(* CODESYS project CtaDevClimaVeneta_1.0.0.0.library
   Description: CtaDevClimaVeneta Library für ClimaVeneta Modbus auslesung
   Version: 1.0.0.0
   Title: CtaDevClimaVeneta
   Author: SIS
   Company: CTA
   DocFormat: reStructuredText
   Placeholder: CtaDevClimaVeneta
   CompiledLibraryCompatibilityVersion: CODESYS V3.5 SP16 Patch 3
   LanguageModelAttribute: qualified-access-only
   DefaultNamespace: CtaDevClimaVeneta

Project tree, tasks and I/O mapping:
  libraries: CtaAppBmk, 2.0.0.1 (CTA); CtaAppReport, 2.0.0.2 (CTA); CtaAppInfluxLog, 1.0.0.1 (CTA); Standard, 3.5.18.0 (System); CtaAppRefrigants, 1.0.0.0 (CTA); CtaAppModbus, 2.0.0.3 (CTA)
  40 Visualizations/
  30 Program Organization Units/
    MODBUS_FB_CLIMAVENETA/
      function block MODBUS_CLIMAVENETA [ST]: COM_DATA
      text list txtAlamsW3000
      text list txtWpReport
  00000000-0000-0000-0000-000000000000|D:\CoDeSys\LibrariesV3\trunk\Intern\CAA\CAA Template\3.4.0.0 draft\Placeholder.xml
  00000000-0000-0000-0000-000000000000|D:\CoDeSys\LibrariesV3\trunk\Intern\CAA\CAA Template\3.2.0.3 draft\Prefix.pdf
  00000000-0000-0000-0000-000000000000|D:\CoDeSys\LibrariesV3\trunk\Intern\CAA\CAA Template\3.5.2.0 draft\Placeholder.xml
  20 Structs/
  50 Images/
  10 Documenation/
    global variables VersionHistory
    global variables readMe
  21 Interface/
  11 Library Parameter/
  12 Konstanten/
  60 Textlisten/
  13 Globale Variablen/
*)

// 10 Documenation/VersionHistory
(* 

.. image:: ../../Images/CTA_Logo.jpg
   :align: right
   :width: 15% 

**Vorlage**   


============ =========== =========== ============================================
**Date**     **Version** **Author**  **Change**
------------ ----------- ----------- --------------------------------------------
22.07.2026   1.0.0.0     SIS         Bibliothek erstellt

============ =========== =========== ============================================


*)
VAR_GLOBAL
    stInfo : STRING:= '0.0.0.0, CtaDevClimaVeneta, CTA';
END_VAR

// 10 Documenation/readMe
(*
**ReadMe**

 
 |  Diese Bibliothek dient der standartisierten auslesung von Climaveneta Maschinen
 |     
*)

VAR_GLOBAL
    xReadMeDone              :   BOOL;
END_VAR

// 30 Program Organization Units/MODBUS_FB_CLIMAVENETA/MODBUS_CLIMAVENETA
FUNCTION_BLOCK MODBUS_CLIMAVENETA
VAR CONSTANT
	stTxtReportError		:	STRING											:= 'CtaDevClimaVeneta.txtWpReport';
END_VAR
VAR_INPUT
	ITF_BMK					:	CtaAppBmk.ITF_BMK;
	ITF_REPORTMANAGER		:	CtaAppReport.ITF_REPORTMANAGER;
	set_point				:	REAL;											// Sollwert
	_rBeschränkung			:	REAL;											// Demand Limit
	_xBeschränkungEN		:	BOOL;											// Demand Limit enable
END_VAR
VAR_OUTPUT
	_xModBusError			:	BOOL;
	_v1k1_on				:	BOOL;
	_v1k2_on				:	BOOL;	
	_v2k1_on				:	BOOL;
	_v2k2_on				:	BOOL;	
	_xAlarm1V1				:	BOOL;
	_xAlarm1V2				:	BOOL;
	_xAlarm1V3				:	BOOL;
	_xAlarm1V4				:	BOOL;
	
	_rHochdruckV1			:	REAL;
	_rHochdruckTempV1		:	REAL;
	_rHochdruckV2			:	REAL;
	_rHochdruckTempV2		:	REAL;
	
	_rNiederdruckV1			:	REAL;
	_rNiederdruckTempV1		:	REAL;
	_rNiederdruckV2			:	REAL;
	_rNiederdruckTempV2		:	REAL;

	_rFehlerCode			:	REAL;
	
END_VAR
VAR
	_ayMbData				:	ARRAY[0..16] OF WORD;
	_ayTrendLogBool			:	ARRAY[1..15] OF CtaAppInfluxLog.FB_LOG_NODE_BOOL;
	_ayTrendLogReal			:	ARRAY[1..15] OF CtaAppInfluxLog.FB_LOG_NODE_REAL;
	_ayReports				:	ARRAY[0..00] OF CtaAppReport.fbReporter;
	_ayMbDataBOOL			:	ARRAY[0..16] OF BOOL;
END_VAR

IF __QUERYINTERFACE(ITF_BMK,ITF_BMK) THEN

	_ayTrendLogReal[01].ENABLE 		:= TRUE;
	_ayTrendLogReal[01].KEY	 		:= CONCAT(ITF_BMK.proGetBMK,'_rHochdruckV1');
	_ayTrendLogReal[01].SET_VALUE	:= _rHochdruckV1;
	
	_ayTrendLogReal[02].ENABLE 		:= TRUE;
	_ayTrendLogReal[02].KEY	 		:= CONCAT(ITF_BMK.proGetBMK,'_rHochdruckV2');
	_ayTrendLogReal[02].SET_VALUE	:= _rHochdruckV2;

	_ayTrendLogReal[03].ENABLE 		:= TRUE;
	_ayTrendLogReal[03].KEY	 		:= CONCAT(ITF_BMK.proGetBMK,'_rNiederdruckV1');
	_ayTrendLogReal[03].SET_VALUE	:= _rNiederdruckV1;
	
	_ayTrendLogReal[04].ENABLE 		:= TRUE;
	_ayTrendLogReal[04].KEY	 		:= CONCAT(ITF_BMK.proGetBMK,'_rNiederdruckV2');
	_ayTrendLogReal[04].SET_VALUE	:= _rNiederdruckV2;
	
	_ayTrendLogReal[05].ENABLE 		:= TRUE;
	_ayTrendLogReal[05].KEY	 		:= CONCAT(ITF_BMK.proGetBMK,'_rFehlerCode');
	_ayTrendLogReal[05].SET_VALUE	:= _rFehlerCode;
	
	_ayTrendLogReal[06].ENABLE 		:= TRUE;
	_ayTrendLogReal[06].KEY	 		:= CONCAT(ITF_BMK.proGetBMK,'_rHochdruckTempV1');
	_ayTrendLogReal[06].SET_VALUE	:= _rHochdruckTempV1;
	
	_ayTrendLogReal[07].ENABLE 		:= TRUE;
	_ayTrendLogReal[07].KEY	 		:= CONCAT(ITF_BMK.proGetBMK,'_rHochdruckTempV2');
	_ayTrendLogReal[07].SET_VALUE	:= _rHochdruckTempV2;
	
	_ayTrendLogReal[08].ENABLE 		:= TRUE;
	_ayTrendLogReal[08].KEY	 		:= CONCAT(ITF_BMK.proGetBMK,'_rNiederdruckTempV1');
	_ayTrendLogReal[08].SET_VALUE	:= _rNiederdruckTempV1;
	
	_ayTrendLogReal[09].ENABLE 		:= TRUE;
	_ayTrendLogReal[09].KEY	 		:= CONCAT(ITF_BMK.proGetBMK,'_rNiederdruckTempV2');
	_ayTrendLogReal[09].SET_VALUE	:= _rNiederdruckTempV2;

	_ayTrendLogBool[05].ENABLE 		:= TRUE;
	_ayTrendLogBool[05].KEY	 		:= CONCAT(ITF_BMK.proGetBMK,'_xAlarm1V1');
	_ayTrendLogBool[05].SET_VALUE	:= _xAlarm1V1;

	_ayTrendLogBool[06].ENABLE 		:= TRUE;
	_ayTrendLogBool[06].KEY	 		:= CONCAT(ITF_BMK.proGetBMK,'_xAlarm1V2');
	_ayTrendLogBool[06].SET_VALUE	:= _xAlarm1V2;

	_ayTrendLogBool[07].ENABLE 		:= TRUE;
	_ayTrendLogBool[07].KEY	 		:= CONCAT(ITF_BMK.proGetBMK,'_xAlarm1V3');
	_ayTrendLogBool[07].SET_VALUE	:= _xAlarm1V3;

	_ayTrendLogBool[08].ENABLE 		:= TRUE;
	_ayTrendLogBool[08].KEY	 		:= CONCAT(ITF_BMK.proGetBMK,'_xAlarm1V4');
	_ayTrendLogBool[08].SET_VALUE	:= _xAlarm1V4;	
	
	(* Rechnung Bar zu Temp *)
	_rHochdruckTempV1 	:= CtaAppRefrigants.fcPressToTemp_UserDefined(_rHochdruckV1,CtaAppRefrigants.GVL_REFRIGANTS.FB_COURRENT_REFRIGANT.enGasType,FALSE);
	_rNiederdruckTempV1 := CtaAppRefrigants.fcPressToTemp_UserDefined(_rNiederdruckV1,CtaAppRefrigants.GVL_REFRIGANTS.FB_COURRENT_REFRIGANT.enGasType,FALSE);
	
	_rHochdruckTempV2	:= CtaAppRefrigants.fcPressToTemp_UserDefined(_rHochdruckV2,CtaAppRefrigants.GVL_REFRIGANTS.FB_COURRENT_REFRIGANT.enGasType,FALSE);
	_rNiederdruckTempV2 := CtaAppRefrigants.fcPressToTemp_UserDefined(_rNiederdruckV2,CtaAppRefrigants.GVL_REFRIGANTS.FB_COURRENT_REFRIGANT.enGasType,FALSE);

	IF __QUERYINTERFACE(ITF_REPORTMANAGER,ITF_REPORTMANAGER) THEN
		_ayReports[0].metReport(	xSetReportIn				:=	_xModBusError,
									iReportID					:=  60,
									enReportTypeIn				:=  CtaAppReport.enReportType.Error,
									enReportAcknowledgeTypeIn	:=	CtaAppReport.enReportacknowledgeType.Auto,
									tDelay						:=	T#1M,
									ITF_BMK_IN					:=  ITF_BMK,
									pstReportTextListIn			:=  ADR(stTxtReportError),
									stOptionalReportText		:=  '',
									iRetryTilReportLock			:=  3,
									xResetCount					:=  FALSE,
									tReset						:=  T#24H);
		ITF_REPORTMANAGER.metSyncReporter(_ayReports[0]);
	END_IF;
END_IF;

METHOD COM_DATA
VAR_INPUT
	ITF_MB_CLIENT		:	CtaAppModbus.ITF_CLIENT;
END_VAR
VAR 
	ITF_MB_CLIENT_TCP	:	CtaAppModbus.ITF_MB_CLIENT_TCP;
	ITF_MB_CLIENT_RTU	:	CtaAppModbus.ITF_MB_CLIENT_RTU;
	offset				: 	INT;
END_VAR
// Modbus TCP
IF __QUERYINTERFACE(ITF_MB_CLIENT, ITF_MB_CLIENT_TCP ) THEN	
	// Delet rtu
	IF __QUERYINTERFACE(ITF_MB_CLIENT_RTU, ITF_MB_CLIENT_RTU ) THEN
		ITF_MB_CLIENT_RTU.DESTROY_ALL_JOBS_REQUEST();
		ITF_MB_CLIENT_RTU := 0;
	END_IF;
	
	_xModBusError := ITF_MB_CLIENT_TCP.ERROR;
	offset		  := -1;	
	
	// High pressure transducer
	ITF_MB_CLIENT_TCP.CREATE_JOB( _byMbFunction := 04 ,	_wMbAdress := TO_WORD(  13 + offset ), _pData := ADR(_ayMbData[00]), _wQuantity := 1); _rHochdruckV1				:= TO_REAL(TO_INT(_ayMbData[00])) / 10 ;
	ITF_MB_CLIENT_TCP.CREATE_JOB( _byMbFunction := 04 ,	_wMbAdress := TO_WORD(  14 + offset ), _pData := ADR(_ayMbData[01]), _wQuantity := 1); _rHochdruckV2				:= TO_REAL(TO_INT(_ayMbData[01])) / 10 ;
     
	// Low pressure transducer                                                                
	ITF_MB_CLIENT_TCP.CREATE_JOB( _byMbFunction := 04 ,	_wMbAdress := TO_WORD(  17 + offset ), _pData := ADR(_ayMbData[02]), _wQuantity := 1); _rNiederdruckV1			:= TO_REAL(TO_INT(_ayMbData[02])) / 10 ;
	ITF_MB_CLIENT_TCP.CREATE_JOB( _byMbFunction := 04 ,	_wMbAdress := TO_WORD(  18 + offset ), _pData := ADR(_ayMbData[03]), _wQuantity := 1); _rNiederdruckV2			:= TO_REAL(TO_INT(_ayMbData[03])) / 10 ;
        
	// Compressor status                                                            
	ITF_MB_CLIENT_TCP.CREATE_JOB( _byMbFunction := 04 ,	_wMbAdress := TO_WORD(5017 + offset ), _pData := ADR(_ayMbData[04]), _wQuantity := 1); _xAlarm1V1	 		:= _ayMbData[04].04;	_v1k1_on		:= _ayMbData[04].2;	
	ITF_MB_CLIENT_TCP.CREATE_JOB( _byMbFunction := 04 ,	_wMbAdress := TO_WORD(5018 + offset ), _pData := ADR(_ayMbData[05]), _wQuantity := 1); _xAlarm1V2	 		:= _ayMbData[05].04;	_v1k2_on		:= _ayMbData[05].2;	
	ITF_MB_CLIENT_TCP.CREATE_JOB( _byMbFunction := 04 ,	_wMbAdress := TO_WORD(5019 + offset ), _pData := ADR(_ayMbData[06]), _wQuantity := 1); _xAlarm1V3	 		:= _ayMbData[06].04;	_v2k1_on		:= _ayMbData[06].2;	 
	ITF_MB_CLIENT_TCP.CREATE_JOB( _byMbFunction := 04 ,	_wMbAdress := TO_WORD(5020 + offset ), _pData := ADR(_ayMbData[07]), _wQuantity := 1); _xAlarm1V4	 		:= _ayMbData[07].04;	_v2k2_on		:= _ayMbData[07].2;
	
	// Active alarm code (with greater priority)                                                                     
	ITF_MB_CLIENT_TCP.CREATE_JOB( _byMbFunction := 04 ,	_wMbAdress := TO_WORD(5034 + offset ), _pData := ADR(_ayMbData[09]), _wQuantity := 1); _rFehlerCode		:= TO_REAL(TO_INT(_ayMbData[09]))  ;

	// Temperature controller limitation in heat pump
	_ayMbData[12] := TO_WORD(TO_INT(_rBeschränkung * 10));
	ITF_MB_CLIENT_TCP.CREATE_JOB( _byMbFunction := 06, 	_wMbAdress := TO_WORD(5046 + offset ), _pData := ADR(_ayMbData[12]), _wQuantity := 1)  ; 
	
	
	_ayMbDataBOOL[00] := _xBeschränkungEN;
	ITF_MB_CLIENT_TCP.CREATE_JOB( _byMbFunction := 05 ,	_wMbAdress := TO_WORD( 284 + offset ), _pData := ADR(_ayMbDataBOOL[00]), _wQuantity := 1);
	
	// Chiller temperature setpoint 
	_ayMbData[13] := TO_WORD(TO_INT(set_point * 10));
	ITF_MB_CLIENT_TCP.CREATE_JOB( _byMbFunction := 06 , _wMbAdress := TO_WORD( 	 2 + offset ), _pData := ADR(_ayMbData[13]), _wQuantity := 1)  ; 
	
// Modbus RTU
ELSIF __QUERYINTERFACE(ITF_MB_CLIENT, ITF_MB_CLIENT_RTU ) THEN	
	// Delet tcp
	IF __QUERYINTERFACE(ITF_MB_CLIENT_TCP, ITF_MB_CLIENT_TCP ) THEN
		ITF_MB_CLIENT_TCP.DESTROY_ALL_JOBS_REQUEST();
		ITF_MB_CLIENT_TCP := 0;
	END_IF;
	
	_xModBusError := ITF_MB_CLIENT_RTU.ERROR;
	offset		  := 0;		
	
	// High pressure transducer
	ITF_MB_CLIENT_RTU.CREATE_JOB( _byMbFunction := 04 ,	_wMbAdress :=   12 , _pData := ADR(_ayMbData[00]), _wQuantity := 1); _rHochdruckV1				:= TO_REAL(TO_INT(_ayMbData[00])) / 10 ;
	ITF_MB_CLIENT_RTU.CREATE_JOB( _byMbFunction := 04 ,	_wMbAdress :=   13 , _pData := ADR(_ayMbData[01]), _wQuantity := 1); _rHochdruckV2				:= TO_REAL(TO_INT(_ayMbData[01])) / 10 ;
	
	// Low pressure transducer
	ITF_MB_CLIENT_RTU.CREATE_JOB( _byMbFunction := 04 ,	_wMbAdress :=   16 , _pData := ADR(_ayMbData[02]), _wQuantity := 1); _rNiederdruckV1			:= TO_REAL(TO_INT(_ayMbData[02])) / 10 ;
	ITF_MB_CLIENT_RTU.CREATE_JOB( _byMbFunction := 04 ,	_wMbAdress :=   17 , _pData := ADR(_ayMbData[03]), _wQuantity := 1); _rNiederdruckV2			:= TO_REAL(TO_INT(_ayMbData[03])) / 10 ;

	// Compressor status
	ITF_MB_CLIENT_RTU.CREATE_JOB( _byMbFunction := 04 ,	_wMbAdress :=  143 , _pData := ADR(_ayMbData[04]), _wQuantity := 1); _xAlarm1V1	 		:= _ayMbData[04].04;	_v1k1_on		:= _ayMbData[04].2;	
	ITF_MB_CLIENT_RTU.CREATE_JOB( _byMbFunction := 04 ,	_wMbAdress :=  144 , _pData := ADR(_ayMbData[05]), _wQuantity := 1); _xAlarm1V2	 		:= _ayMbData[05].04;	_v1k2_on		:= _ayMbData[05].2;	
	ITF_MB_CLIENT_RTU.CREATE_JOB( _byMbFunction := 04 ,	_wMbAdress :=  145 , _pData := ADR(_ayMbData[06]), _wQuantity := 1); _xAlarm1V3	 		:= _ayMbData[06].04;	_v2k1_on		:= _ayMbData[06].2;	 
	ITF_MB_CLIENT_RTU.CREATE_JOB( _byMbFunction := 04 ,	_wMbAdress :=  146 , _pData := ADR(_ayMbData[07]), _wQuantity := 1); _xAlarm1V4	 		:= _ayMbData[07].04;	_v2k2_on		:= _ayMbData[07].2;
	
	// Active alarm code (with greater priority) 
	ITF_MB_CLIENT_RTU.CREATE_JOB( _byMbFunction := 04 ,	_wMbAdress :=  160 , _pData := ADR(_ayMbData[09]), _wQuantity := 1); _rFehlerCode		:= TO_REAL(TO_INT(_ayMbData[09]))  ;

	// Temperature controller limitation in heat pump
	_ayMbData[12] := TO_WORD(TO_INT(_rBeschränkung * 10));
	ITF_MB_CLIENT_RTU.CREATE_JOB( _byMbFunction := 06, 	_wMbAdress :=  172, _pData := ADR(_ayMbData[12]), _wQuantity := 1)  ; 
	
	_ayMbDataBOOL[00] := _xBeschränkungEN;
	ITF_MB_CLIENT_RTU.CREATE_JOB( _byMbFunction := 05 ,	_wMbAdress :=   33 , _pData := ADR(_ayMbDataBOOL[00]), _wQuantity := 1);
	
	// Chiller temperature setpoint 
	_ayMbData[13] := TO_WORD(TO_INT(set_point * 10));
	ITF_MB_CLIENT_RTU.CREATE_JOB( _byMbFunction := 06 , _wMbAdress :=  	 1, _pData := ADR(_ayMbData[13]), _wQuantity := 1)  ; 
	

ELSE
	_xModBusError := TRUE;
END_IF;
END_METHOD

END_FUNCTION_BLOCK

(* text list txtAlamsW3000 (id | default | de | en | fr | it)
  2 | Phasensequenz / Spannung außer Bereich | Phasensequenz / Spannung außer Bereich | Phase sequence / voltage out of range | Séquence de phases / tension hors plage | Sequenza di fase / tensione fuori intervallo
  3 | Kein Wasserfluss am Verdampfer | Kein Wasserfluss am Verdampfer | No water flow at evaporator | No water flow at évaporateur | No water flow at evaporatore
  5 | Niedrige Temperatur am Eingang | Niedrige Temperatur am Eingang | Low temperature am inlet | Low temperature am entrée | Low temperature am ingresso
  6 | Hohe Temperatur am Eingang | Hohe Temperatur am Eingang | High temperature am inlet | High temperature am entrée | High temperature am ingresso
  7 | Blockierung alternative Quelle der Anlage | Blockierung alternative Quelle der Anlage | Lockout: plant alternative source | Blocage : source alternative de l’installation | Blocco: fonte alternativa dell’impianto
  8 | Blockierung alternative DHW -quelle | Blockierung alternative DHW -quelle | Lockout: alternative DHW source | Blocage : source ECS (DHW) alternative | Blocco: sorgente ACS alternativa
  10 | Frostschutz Verdampfer Niedrige Wassertemperatur am Verdampferausgang. Es wird außerdem angezeigt, für welchen Verdampfer der Alarm gilt (bei mehr als einem Verdampfer). Der Alarm tritt auch dann auf, wenn die Frostschutz - Begrenzung in einem Zeitraum von 8 Betriebsstunden öfter als 5 -mal ausgelöst wird. M CI STG0073 | Frostschutz Verdampfer Niedrige Wassertemperatur am Verdampferausgang. Es wird außerdem angezeigt, für welchen Verdampfer der Alarm gilt (bei mehr als einem Verdampfer). Der Alarm tritt auch dann auf, wenn die Frostschutz - Begrenzung in einem Zeitraum von 8 Betriebsstunden öfter als 5 -mal ausgelöst wird. M CI STG0073 | Frost protection evaporator Niedrige Wassertemperatur am evaporatoroutlet. Es wird außerdem angezeigt, für welchen evaporator Alarm gilt (bei mehr als einem evaporator). Alarm tritt auch dann auf, wenn Frostschutz - Begrenzung in einem Zeitraum von 8 Betriebsstunden öfter als 5 -mal ausgelöst wird. M CI STG0073 | Frost protection évaporateur Niedrige Wassertemperatur am évaporateursortie. Es wird außerdem angezeigt, für welchen évaporateur Alarm gilt (bei mehr als einem évaporateur). Alarm tritt auch dann auf, wenn Frostschutz - Begrenzung in einem Zeitraum von 8 Betriebsstunden öfter als 5 -mal ausgelöst wird. M CI STG0073 | Frost protection evaporatore Niedrige Wassertemperatur am evaporatoreuscita. Es wird außerdem angezeigt, für welchen evaporatore Alarm gilt (bei mehr als einem evaporatore). Alarm tritt auch dann auf, wenn Frostschutz - Begrenzung in einem Zeitraum von 8 Betriebsstunden öfter als 5 -mal ausgelöst wird. M CI STG0073
  14 | Unzureichender Anlagendruck | Unzureichender Anlagendruck | Insufficient system pressure | Pression système insuffisante | Pressione impianto insufficiente
  17 | Niedrige Außenlufttemperatur | Niedrige Außenlufttemperatur | Low outdoor air temperature | Température extérieure basse | Temperatura aria esterna bassa
  21 | Geringe Wassermenge in der Anlage | Geringe Wassermenge in der Anlage | Low water content in system | Faible volume d’eau dans l’installation | Basso contenuto d’acqua nel sistema
  22 | Niedriger Wasserdurchfluss in der Anlage | Niedriger Wasserdurchfluss in der Anlage | Low water flow in system | Low water flow in installation | Low water flow in impianto
  23 | Hoher Wasserdurchfluss | Hoher Wasserdurchfluss | High water flow | Débit d’eau élevé | Portata d’acqua elevata
  41 | Niedrige Temperatur am Verflüssigereingang | Niedrige Temperatur am Verflüssigereingang | Low temperature at condenser inlet | Low temperature at condenser inlet | Low temperature at condenser inlet
  42 | Hohe Temperatur am Verflüssigerausgang | Hohe Temperatur am Verflüssigerausgang | High temperature at condenser outlet | High temperature at condenser outlet | High temperature at condenser outlet
  43 | Niedriger Wasserdurchfluss im Verflüssiger | Niedriger Wasserdurchfluss im Verflüssiger | Low water flow im condenser | Low water flow im condenseur | Low water flow im condensatore
  44 | Hoher Wasserdurchfluss im Verflüssiger | Hoher Wasserdurchfluss im Verflüssiger | High water flow | Débit d’eau élevé | Portata d’acqua elevata
  45 | Kein Wasserfluss am Verflüssiger „Kein Wasserfluss am Verdampfer” (nur bei Wasser/Wasser -Einheiten mit Freon -Umkehr). A/M U | Kein Wasserfluss am Verflüssiger „Kein Wasserfluss am Verdampfer” (nur bei Wasser/Wasser -Einheiten mit Freon -Umkehr). A/M U | No water flow at condenser „No water flow at evaporator” (nur bei Wasser/Wasser -uniten mit Freon -Umkehr). A/M U | No water flow at condenseur „No water flow at évaporateur” (nur bei Wasser/Wasser -unitéen mit Freon -Umkehr). A/M U | No water flow at condensatore „No water flow at evaporatore” (nur bei Wasser/Wasser -unitàen mit Freon -Umkehr). A/M U
  46 | Kein Wasserfluss am WRG | Kein Wasserfluss am WRG | No water flow at heat recovery | No water flow at récupération de chaleur | No water flow at recupero di calore
  50 | Totalausfall Kältemaschine  | Totalausfall Kältemaschine  | Complete failure of the cooling system | Panne complète du système de refroidissement | Guasto completo della macchina frigorifera
  51 | Wartung Pumpe 1 | Wartung Pumpe 1 | Maintenance pump 1 | Maintenance pompe 1 | Maintenance pompa 1
  57 | Wartung WRG/DHW -Pumpe (Bei Einheiten mit WRG -Pumpe) Die Grenze der zulässigen Stunden der WRG -Pumpe wurde überschritten. S - STG0007 | Wartung WRG/DHW -Pumpe (Bei Einheiten mit WRG -Pumpe) Die Grenze der zulässigen Stunden der WRG -Pumpe wurde überschritten. S - STG0007 | Maintenance heat recovery/DHW -pump (Bei uniten mit heat recovery -pump) Grenze zulässigen Stunden heat recovery -pump wurde überschritten. S - STG0007 | Maintenance récupération de chaleur/DHW -pompe (Bei unitéen mit récupération de chaleur -pompe) Grenze zulässigen Stunden récupération de chaleur -pompe wurde überschritten. S - STG0007 | Maintenance recupero di calore/DHW -pompa (Bei unitàen mit recupero di calore -pompa) Grenze zulässigen Stunden recupero di calore -pompa wurde überschritten. S - STG0007
  58 | Wartung Verflüssigerpumpe (Bei Einheiten mit Verflüssigerpumpe) Die Grenze der zulässigen Stunden der Verflüssigerpumpe wurde überschritten. S - STG0010 | Wartung Verflüssigerpumpe (Bei Einheiten mit Verflüssigerpumpe) Die Grenze der zulässigen Stunden der Verflüssigerpumpe wurde überschritten. S - STG0010 | Maintenance condenserpump (Bei uniten mit condenserpump) Grenze zulässigen Stunden condenserpump wurde überschritten. S - STG0010 | Maintenance condenseurpompe (Bei unitéen mit condenseurpompe) Grenze zulässigen Stunden condenseurpompe wurde überschritten. S - STG0010 | Maintenance condensatorepompa (Bei unitàen mit condensatorepompa) Grenze zulässigen Stunden condensatorepompa wurde überschritten. S - STG0010
  61 | Offline Driver Unterkühlung / erste Stufe Nr.1 | Offline Driver Unterkühlung / erste Stufe Nr.1 | Offline Driver Unterkühlung / erste Stufe Nr.1 | Offline Driver Unterkühlung / erste Stufe Nr.1 | Offline Driver Unterkühlung / erste Stufe Nr.1
  62 | Offline Driver Unterkühlung / erste Stufe Nr.2 „Wie oben, für den Kreislauf Nr.2“ / Ventil erste Stufe des Verdichters 2. A CI | Offline Driver Unterkühlung / erste Stufe Nr.2 „Wie oben, für den Kreislauf Nr.2“ / Ventil erste Stufe des Verdichters 2. A CI | Offline Driver Unterkühlung / erste Stufe Nr.2 „Wie oben, für circuit Nr.2“ / Ventil erste Stufe compressors 2. A CI | Offline Driver Unterkühlung / erste Stufe Nr.2 „Wie oben, für circuit Nr.2“ / Ventil erste Stufe compresseurs 2. A CI | Offline Driver Unterkühlung / erste Stufe Nr.2 „Wie oben, für circuito Nr.2“ / Ventil erste Stufe compressores 2. A CI
  63 | Offline Driver Unterkühlung / erste Stufe Nr.3 „Wie oben, für den Kreislauf Nr.1“ / Ventil erste Stufe des Verdichters 3. A CI | Offline Driver Unterkühlung / erste Stufe Nr.3 „Wie oben, für den Kreislauf Nr.1“ / Ventil erste Stufe des Verdichters 3. A CI | Offline Driver Unterkühlung / erste Stufe Nr.3 „Wie oben, für circuit Nr.1“ / Ventil erste Stufe compressors 3. A CI | Offline Driver Unterkühlung / erste Stufe Nr.3 „Wie oben, für circuit Nr.1“ / Ventil erste Stufe compresseurs 3. A CI | Offline Driver Unterkühlung / erste Stufe Nr.3 „Wie oben, für circuito Nr.1“ / Ventil erste Stufe compressores 3. A CI
  64 | Offline Driver Unterkühlung / erste Stufe Nr.4 „Wie oben, für den Kreislauf Nr.2“ / Ventil erste Stufe des Verdichters 4. A CI | Offline Driver Unterkühlung / erste Stufe Nr.4 „Wie oben, für den Kreislauf Nr.2“ / Ventil erste Stufe des Verdichters 4. A CI | Offline Driver Unterkühlung / erste Stufe Nr.4 „Wie oben, für circuit Nr.2“ / Ventil erste Stufe compressors 4. A CI | Offline Driver Unterkühlung / erste Stufe Nr.4 „Wie oben, für circuit Nr.2“ / Ventil erste Stufe compresseurs 4. A CI | Offline Driver Unterkühlung / erste Stufe Nr.4 „Wie oben, für circuito Nr.2“ / Ventil erste Stufe compressores 4. A CI
  65 | Niedrige Wassermenge im Wärmerückgewinnungskreislauf | Niedrige Wassermenge im Wärmerückgewinnungskreislauf | Niedrige Wassermenge im heat recovery circuit | Niedrige Wassermenge im circuit de récupération de chaleur | Niedrige Wassermenge im circuit di recupero di calore
  66 | Niedriger Wasserdurchfluss im Wärmerückgewinnungskreislauf | Niedriger Wasserdurchfluss im Wärmerückgewinnungskreislauf | Low water flow im heat recovery circuit | Low water flow im circuit de récupération de chaleur | Low water flow im circuit di recupero di calore
  67 | Alarm Antilegionellenfunktion | Alarm Antilegionellenfunktion | Alarm Antilegionellenfunktion | Alarm Antilegionellenfunktion | Alarm Antilegionellenfunktion
  68 | Störung von Steuerung Kühlteil Meldet einen von der Hauptreglereinheit kommenden Alarm in den Einheiten mit +2P -Modul. Um den Alarm im Detail anzuzeigen und rückzustellen, muss mit der Tastenkombination [ESC+UP] zur Schnittstelle der Hauptreglereinheit übergegangen werden. S - | Störung von Steuerung Kühlteil Meldet einen von der Hauptreglereinheit kommenden Alarm in den Einheiten mit +2P -Modul. Um den Alarm im Detail anzuzeigen und rückzustellen, muss mit der Tastenkombination [ESC+UP] zur Schnittstelle der Hauptreglereinheit übergegangen werden. S - | Fault von Steuerung Kühlteil Meldet einen von Hauptreglerunit kommenden Alarm in uniten mit +2P -Modul. Um Alarm im Detail anzuzeigen und rückzustellen, muss mit Tastenkombination [ESC+UP] zur Schnittstelle Hauptreglerunit übergegangen werden. S - | Fault von Steuerung Kühlteil Meldet einen von Hauptreglerunité kommenden Alarm in unitéen mit +2P -Modul. Um Alarm im Detail anzuzeigen und rückzustellen, muss mit Tastenkombination [ESC+UP] zur Schnittstelle Hauptreglerunité übergegangen werden. S - | Fault von Steuerung Kühlteil Meldet einen von Hauptreglerunità kommenden Alarm in unitàen mit +2P -Modul. Um Alarm im Detail anzuzeigen und rückzustellen, muss mit Tastenkombination [ESC+UP] zur Schnittstelle Hauptreglerunità übergegangen werden. S -
  69 | Störung von Steuerung Luftteil Meldet einen von der Steuerung des Luftteils kommenden Alarm in den Rooftop -Einheiten. Um den Alarm im Detail anzuzeigen und rückzustellen, muss mit der Tastenkombination [ESC+UP] zur Schnittstelle der Hauptreglereinheit übergegangen werden. S - | Störung von Steuerung Luftteil Meldet einen von der Steuerung des Luftteils kommenden Alarm in den Rooftop -Einheiten. Um den Alarm im Detail anzuzeigen und rückzustellen, muss mit der Tastenkombination [ESC+UP] zur Schnittstelle der Hauptreglereinheit übergegangen werden. S - | Fault von Steuerung Luftteil Meldet einen von Steuerung Luftteils kommenden Alarm in Rooftop -uniten. Um Alarm im Detail anzuzeigen und rückzustellen, muss mit Tastenkombination [ESC+UP] zur Schnittstelle Hauptreglerunit übergegangen werden. S - | Fault von Steuerung Luftteil Meldet einen von Steuerung Luftteils kommenden Alarm in Rooftop -unitéen. Um Alarm im Detail anzuzeigen und rückzustellen, muss mit Tastenkombination [ESC+UP] zur Schnittstelle Hauptreglerunité übergegangen werden. S - | Fault von Steuerung Luftteil Meldet einen von Steuerung Luftteils kommenden Alarm in Rooftop -unitàen. Um Alarm im Detail anzuzeigen und rückzustellen, muss mit Tastenkombination [ESC+UP] zur Schnittstelle Hauptreglerunità übergegangen werden. S -
  70 | Störung von Steuerung +2P -Modul Meldet einen von der Reglereinheit kommenden Alarm des Moduls +2P. Um den Alarm im Detail anzuzeigen und rückzustellen, muss mit der Tastenkombination [ESC+UP] zur Schnittstelle der Reglereinheit +2P übergegangen werden. S - | Störung von Steuerung +2P -Modul Meldet einen von der Reglereinheit kommenden Alarm des Moduls +2P. Um den Alarm im Detail anzuzeigen und rückzustellen, muss mit der Tastenkombination [ESC+UP] zur Schnittstelle der Reglereinheit +2P übergegangen werden. S - | Fault von Steuerung +2P -Modul Meldet einen von Reglerunit kommenden Alarm Moduls +2P. Um Alarm im Detail anzuzeigen und rückzustellen, muss mit Tastenkombination [ESC+UP] zur Schnittstelle Reglerunit +2P übergegangen werden. S - | Fault von Steuerung +2P -Modul Meldet einen von Reglerunité kommenden Alarm Moduls +2P. Um Alarm im Detail anzuzeigen und rückzustellen, muss mit Tastenkombination [ESC+UP] zur Schnittstelle Reglerunité +2P übergegangen werden. S - | Fault von Steuerung +2P -Modul Meldet einen von Reglerunità kommenden Alarm Moduls +2P. Um Alarm im Detail anzuzeigen und rückzustellen, muss mit Tastenkombination [ESC+UP] zur Schnittstelle Reglerunità +2P übergegangen werden. S -
  72 | Hoher Wasserdurchfluss im Wärmerückgewinnungskreislauf | Hoher Wasserdurchfluss im Wärmerückgewinnungskreislauf | High water flow | Débit d’eau élevé | Portata d’acqua elevata
  75 | Frostschutz Verflüssiger Niedrige Wassertemperatur am Ausgang des Verflüssigers. Mit Ausnahme von W3000+ Basis wird außerdem angegeben, welcher Verflüssiger (bei mehr als einem) von dem Alarm betroffen ist. Der Alarm tritt auch dann auf, wenn die Frostschutzfunktion mehr als 5 -mal innerhalb von 8 Betriebsstunden ausgelöst wird (nur bei Wasser/Wasser -Einheiten mit Freon -Umkehr). M U* STG0077 | Frostschutz Verflüssiger Niedrige Wassertemperatur am Ausgang des Verflüssigers. Mit Ausnahme von W3000+ Basis wird außerdem angegeben, welcher Verflüssiger (bei mehr als einem) von dem Alarm betroffen ist. Der Alarm tritt auch dann auf, wenn die Frostschutzfunktion mehr als 5 -mal innerhalb von 8 Betriebsstunden ausgelöst wird (nur bei Wasser/Wasser -Einheiten mit Freon -Umkehr). M U* STG0077 | Frost protection condenser Niedrige Wassertemperatur am outlet condensers. Mit Ausnahme von W3000+ Basis wird außerdem angegeben, welcher condenser (bei mehr als einem) von Alarm betroffen ist. Alarm tritt auch dann auf, wenn Frostschutzfunktion mehr als 5 -mal innerhalb von 8 Betriebsstunden ausgelöst wird (nur bei Wasser/Wasser -uniten mit Freon -Umkehr). M U* STG0077 | Frost protection condenseur Niedrige Wassertemperatur am sortie condenseurs. Mit Ausnahme von W3000+ Basis wird außerdem angegeben, welcher condenseur (bei mehr als einem) von Alarm betroffen ist. Alarm tritt auch dann auf, wenn Frostschutzfunktion mehr als 5 -mal innerhalb von 8 Betriebsstunden ausgelöst wird (nur bei Wasser/Wasser -unitéen mit Freon -Umkehr). M U* STG0077 | Frost protection condensatore Niedrige Wassertemperatur am uscita condensatores. Mit Ausnahme von W3000+ Basis wird außerdem angegeben, welcher condensatore (bei mehr als einem) von Alarm betroffen ist. Alarm tritt auch dann auf, wenn Frostschutzfunktion mehr als 5 -mal innerhalb von 8 Betriebsstunden ausgelöst wird (nur bei Wasser/Wasser -unitàen mit Freon -Umkehr). M U* STG0077
  76 | Frostschutz WRG Niedrige Temperatur des Wassers am Ausgang des WRG. A U* STG0079 | Frostschutz WRG Niedrige Temperatur des Wassers am Ausgang des WRG. A U* STG0079 | Frost protection heat recovery Low temperature Wassers am outlet heat recovery. A U* STG0079 | Frost protection récupération de chaleur Low temperature Wassers am sortie récupération de chaleur. A U* STG0079 | Frost protection recupero di calore Low temperature Wassers am uscita recupero di calore. A U* STG0079
  79 | Anlagen -Steuermodul VPF nicht angeschlossen Das Modul für die Wasserdurchflussregelung am Primärkreis ist nicht angeschlossen. A - | Anlagen -Steuermodul VPF nicht angeschlossen Das Modul für die Wasserdurchflussregelung am Primärkreis ist nicht angeschlossen. A - | systemn -Steuermodul VPF nicht angeschlossen Modul für Wasserdurchflussregelung am Primärkreis ist nicht angeschlossen. A - | installationn -Steuermodul VPF nicht angeschlossen Modul für Wasserdurchflussregelung am Primärkreis ist nicht angeschlossen. A - | impianton -Steuermodul VPF nicht angeschlossen Modul für Wasserdurchflussregelung am Primärkreis ist nicht angeschlossen. A -
  80 | Störung Anlagen -Steuermodul VPF Am Modul für die Wasserdurchflussregelung am Primärkreis ist eine Störung aufgetreten. Die Störung an der Benutzerschnittstelle des Moduls überprüfen. A - | Störung Anlagen -Steuermodul VPF Am Modul für die Wasserdurchflussregelung am Primärkreis ist eine Störung aufgetreten. Die Störung an der Benutzerschnittstelle des Moduls überprüfen. A - | Fault systemn -Steuermodul VPF Am Modul für Wasserdurchflussregelung am Primärkreis ist eine Störung aufgetreten. Störung an Benutzerschnittstelle Moduls überprüfen. A - | Fault installationn -Steuermodul VPF Am Modul für Wasserdurchflussregelung am Primärkreis ist eine Störung aufgetreten. Störung an Benutzerschnittstelle Moduls überprüfen. A - | Fault impianton -Steuermodul VPF Am Modul für Wasserdurchflussregelung am Primärkreis ist eine Störung aufgetreten. Störung an Benutzerschnittstelle Moduls überprüfen. A -
  81 | Schutzschalter Pumpe 1 | Schutzschalter Pumpe 1 | Protection switch pump 1 | Protection switch pompe 1 | Protection switch pompa 1
  82 | Schutzschalter Pumpe 2 (Bei Einheiten mit mehr als einer Pumpe) weist diese Meldung auf die Überhitzung der Pumpe 2 hin. M U* | Schutzschalter Pumpe 2 (Bei Einheiten mit mehr als einer Pumpe) weist diese Meldung auf die Überhitzung der Pumpe 2 hin. M U* | Protection switch pump 2 (Bei uniten mit mehr als einer pump) weist diese Meldung auf Überhitzung pump 2 hin. M U* | Protection switch pompe 2 (Bei unitéen mit mehr als einer pompe) weist diese Meldung auf Überhitzung pompe 2 hin. M U* | Protection switch pompa 2 (Bei unitàen mit mehr als einer pompa) weist diese Meldung auf Überhitzung pompa 2 hin. M U*
  85 | Schutzschalter Verflüssigerpumpe | Schutzschalter Verflüssigerpumpe | Protection switch condenserpump | Protection switch condenseurpompe | Protection switch condensatorepompa
  86 | Schutzschalter WRG | Schutzschalter WRG | Protection switch heat recovery | Protection switch récupération de chaleur | Protection switch recupero di calore
  87 | Schutzschalter Glykolpumpe | Schutzschalter Glykolpumpe | Protection switch glycol pump | Protection switch pompe glycol | Protection switch pompa glicole
  90 | Slave nicht angeschlossen | Slave nicht angeschlossen | Slave nicht angeschlossen | Slave nicht angeschlossen | Slave nicht angeschlossen
  91 | Trennung Expansion 1 Meldet, dass die Expansion Nr. 1 des Masters nicht angeschlossen ist	 die Meldung Master erscheint bei Einheiten mit 3 oder 4 Kreisläufen. A U | Trennung Expansion 1 Meldet, dass die Expansion Nr. 1 des Masters nicht angeschlossen ist	 die Meldung Master erscheint bei Einheiten mit 3 oder 4 Kreisläufen. A U | Disconnection Expansion 1 Meldet, dass Expansion Nr. 1 Masters nicht angeschlossen ist	 Meldung Master erscheint bei uniten mit 3 oder 4 Kreisläufen. A U | Disconnection Expansion 1 Meldet, dass Expansion Nr. 1 Masters nicht angeschlossen ist	 Meldung Master erscheint bei unitéen mit 3 oder 4 Kreisläufen. A U | Disconnection Expansion 1 Meldet, dass Expansion Nr. 1 Masters nicht angeschlossen ist	 Meldung Master erscheint bei unitàen mit 3 oder 4 Kreisläufen. A U
  92 | Trennung Expansion 2 „Wie oben, für Expansion Nr.2“ A U | Trennung Expansion 2 „Wie oben, für Expansion Nr.2“ A U | Disconnection Expansion 2 „Wie oben, für Expansion Nr.2“ A U | Disconnection Expansion 2 „Wie oben, für Expansion Nr.2“ A U | Disconnection Expansion 2 „Wie oben, für Expansion Nr.2“ A U
  93 | Trennung Expansion 3 „Wie oben, für Expansion Nr.3“ A U | Trennung Expansion 3 „Wie oben, für Expansion Nr.3“ A U | Disconnection Expansion 3 „Wie oben, für Expansion Nr.3“ A U | Disconnection Expansion 3 „Wie oben, für Expansion Nr.3“ A U | Disconnection Expansion 3 „Wie oben, für Expansion Nr.3“ A U
  94 | Trennung Expansion 4 „Wie oben, für Expansion Nr.4“ A U | Trennung Expansion 4 „Wie oben, für Expansion Nr.4“ A U | Disconnection Expansion 4 „Wie oben, für Expansion Nr.4“ A U | Disconnection Expansion 4 „Wie oben, für Expansion Nr.4“ A U | Disconnection Expansion 4 „Wie oben, für Expansion Nr.4“ A U
  95 | Trennung Expansion 5 „Wie oben, für Expansion Nr.5“ A U | Trennung Expansion 5 „Wie oben, für Expansion Nr.5“ A U | Disconnection Expansion 5 „Wie oben, für Expansion Nr.5“ A U | Disconnection Expansion 5 „Wie oben, für Expansion Nr.5“ A U | Disconnection Expansion 5 „Wie oben, für Expansion Nr.5“ A U
  100 | Energiezähler nicht angeschlossen | Energiezähler nicht angeschlossen | Energy meter not connected | Compteur d’énergie non connecté | Contatore di energia non collegato
  101 | Trennung Expansion 1 Slave | Trennung Expansion 1 Slave | Disconnection Expansion 1 Slave | Disconnection Expansion 1 Slave | Disconnection Expansion 1 Slave
  102 | Trennung Expansion 2 Slave „Wie oben, für Expansion Nr.2“ A U | Trennung Expansion 2 Slave „Wie oben, für Expansion Nr.2“ A U | Disconnection Expansion 2 Slave „Wie oben, für Expansion Nr.2“ A U | Disconnection Expansion 2 Slave „Wie oben, für Expansion Nr.2“ A U | Disconnection Expansion 2 Slave „Wie oben, für Expansion Nr.2“ A U
  103 | Trennung Expansion 3 Slave „Wie oben, für Expansion Nr.3“ A U | Trennung Expansion 3 Slave „Wie oben, für Expansion Nr.3“ A U | Disconnection Expansion 3 Slave „Wie oben, für Expansion Nr.3“ A U | Disconnection Expansion 3 Slave „Wie oben, für Expansion Nr.3“ A U | Disconnection Expansion 3 Slave „Wie oben, für Expansion Nr.3“ A U
  104 | Trennung Expansion 4 Slave „Wie oben, für Expansion Nr.4“ A U | Trennung Expansion 4 Slave „Wie oben, für Expansion Nr.4“ A U | Disconnection Expansion 4 Slave „Wie oben, für Expansion Nr.4“ A U | Disconnection Expansion 4 Slave „Wie oben, für Expansion Nr.4“ A U | Disconnection Expansion 4 Slave „Wie oben, für Expansion Nr.4“ A U
  105 | Trennung Expansion 5 Slave „Wie oben, für Expansion Nr.5“ A U | Trennung Expansion 5 Slave „Wie oben, für Expansion Nr.5“ A U | Disconnection Expansion 5 Slave „Wie oben, für Expansion Nr.5“ A U | Disconnection Expansion 5 Slave „Wie oben, für Expansion Nr.5“ A U | Disconnection Expansion 5 Slave „Wie oben, für Expansion Nr.5“ A U
  106 | Trennung P3 -Modul | Trennung P3 -Modul | Disconnection P3 -Modul | Disconnection P3 -Modul | Disconnection P3 -Modul
  111 | Öl Verdichter 1 | Öl Verdichter 1 | Öl compressor 1 | Öl compresseur 1 | Öl compressore 1
  112 | Öl Verdichter 2 „Wie oben, für den Verdichter Nr.2“. A/M CO | Öl Verdichter 2 „Wie oben, für den Verdichter Nr.2“. A/M CO | Öl compressor 2 „Wie oben, für compressor Nr.2“. A/M CO | Öl compresseur 2 „Wie oben, für compresseur Nr.2“. A/M CO | Öl compressore 2 „Wie oben, für compressore Nr.2“. A/M CO
  113 | Öl Verdichter 3 „Wie oben, für den Verdichter Nr.3“. A/M CO | Öl Verdichter 3 „Wie oben, für den Verdichter Nr.3“. A/M CO | Öl compressor 3 „Wie oben, für compressor Nr.3“. A/M CO | Öl compresseur 3 „Wie oben, für compresseur Nr.3“. A/M CO | Öl compressore 3 „Wie oben, für compressore Nr.3“. A/M CO
  114 | Öl Verdichter 4 „Wie oben, für den Verdichter Nr.4“. A/M CO | Öl Verdichter 4 „Wie oben, für den Verdichter Nr.4“. A/M CO | Öl compressor 4 „Wie oben, für compressor Nr.4“. A/M CO | Öl compresseur 4 „Wie oben, für compresseur Nr.4“. A/M CO | Öl compressore 4 „Wie oben, für compressore Nr.4“. A/M CO
  121 | Hohe Austrittstemperatur Verdichter 1 | Hohe Austrittstemperatur Verdichter 1 | Hohe Austrittstemperatur compressor 1 | Hohe Austrittstemperatur compresseur 1 | Hohe Austrittstemperatur compressore 1
  122 | Hohe Austrittstemperatur Verdichter 2 „Wie oben, für den Verdichter Nr.2“. A/M CO | Hohe Austrittstemperatur Verdichter 2 „Wie oben, für den Verdichter Nr.2“. A/M CO | Hohe Austrittstemperatur compressor 2 „Wie oben, für compressor Nr.2“. A/M CO | Hohe Austrittstemperatur compresseur 2 „Wie oben, für compresseur Nr.2“. A/M CO | Hohe Austrittstemperatur compressore 2 „Wie oben, für compressore Nr.2“. A/M CO
  123 | Hohe Austrittstemperatur Verdichter 3 „Wie oben, für den Verdichter Nr.3“. A/M CO | Hohe Austrittstemperatur Verdichter 3 „Wie oben, für den Verdichter Nr.3“. A/M CO | Hohe Austrittstemperatur compressor 3 „Wie oben, für compressor Nr.3“. A/M CO | Hohe Austrittstemperatur compresseur 3 „Wie oben, für compresseur Nr.3“. A/M CO | Hohe Austrittstemperatur compressore 3 „Wie oben, für compressore Nr.3“. A/M CO
  124 | Hohe Austrittstemperatur Verdichter 4 „Wie oben, für den Verdichter Nr.4“. A/M CO | Hohe Austrittstemperatur Verdichter 4 „Wie oben, für den Verdichter Nr.4“. A/M CO | Hohe Austrittstemperatur compressor 4 „Wie oben, für compressor Nr.4“. A/M CO | Hohe Austrittstemperatur compresseur 4 „Wie oben, für compresseur Nr.4“. A/M CO | Hohe Austrittstemperatur compressore 4 „Wie oben, für compressore Nr.4“. A/M CO
  125 | Hohe Austrittstemperatur Verdichter 5 „Wie oben, für den Verdichter Nr. 5“. A/M CO | Hohe Austrittstemperatur Verdichter 5 „Wie oben, für den Verdichter Nr. 5“. A/M CO | Hohe Austrittstemperatur compressor 5 „Wie oben, für compressor Nr. 5“. A/M CO | Hohe Austrittstemperatur compresseur 5 „Wie oben, für compresseur Nr. 5“. A/M CO | Hohe Austrittstemperatur compressore 5 „Wie oben, für compressore Nr. 5“. A/M CO
  126 | Hohe Austrittstemperatur Verdichter 6 „Wie oben, für den Verdichter Nr. 6“. A/M CO | Hohe Austrittstemperatur Verdichter 6 „Wie oben, für den Verdichter Nr. 6“. A/M CO | Hohe Austrittstemperatur compressor 6 „Wie oben, für compressor Nr. 6“. A/M CO | Hohe Austrittstemperatur compresseur 6 „Wie oben, für compresseur Nr. 6“. A/M CO | Hohe Austrittstemperatur compressore 6 „Wie oben, für compressore Nr. 6“. A/M CO
  127 | Hohe Austrittstemperatur Verdichter 7 „Wie oben, für den Verdichter Nr. 7“. A/M CO | Hohe Austrittstemperatur Verdichter 7 „Wie oben, für den Verdichter Nr. 7“. A/M CO | Hohe Austrittstemperatur compressor 7 „Wie oben, für compressor Nr. 7“. A/M CO | Hohe Austrittstemperatur compresseur 7 „Wie oben, für compresseur Nr. 7“. A/M CO | Hohe Austrittstemperatur compressore 7 „Wie oben, für compressore Nr. 7“. A/M CO
  128 | Hohe Austrittstemperatur Verdichter 8 „Wie oben, für den Verdichter Nr. 8“. A/M CO | Hohe Austrittstemperatur Verdichter 8 „Wie oben, für den Verdichter Nr. 8“. A/M CO | Hohe Austrittstemperatur compressor 8 „Wie oben, für compressor Nr. 8“. A/M CO | Hohe Austrittstemperatur compresseur 8 „Wie oben, für compresseur Nr. 8“. A/M CO | Hohe Austrittstemperatur compressore 8 „Wie oben, für compressore Nr. 8“. A/M CO
  131 | Störung Verdichter 1 | Störung Verdichter 1 | Fault compressor 1 | Fault compresseur 1 | Fault compressore 1
  132 | Störung Verdichter 2 „Wie oben, für den Verdichter Low Lift -Pumpe Nr.2“. M - A/M CO | Störung Verdichter 2 „Wie oben, für den Verdichter Low Lift -Pumpe Nr.2“. M - A/M CO | Fault compressor 2 „Wie oben, für compressor Low Lift -pump Nr.2“. M - A/M CO | Fault compresseur 2 „Wie oben, für compresseur Low Lift -pompe Nr.2“. M - A/M CO | Fault compressore 2 „Wie oben, für compressore Low Lift -pompa Nr.2“. M - A/M CO
  133 | Störung Verdichter 3 „Wie oben, für den Verdichter Low Lift -Pumpe Nr.3“. M - A/M CO | Störung Verdichter 3 „Wie oben, für den Verdichter Low Lift -Pumpe Nr.3“. M - A/M CO | Fault compressor 3 „Wie oben, für compressor Low Lift -pump Nr.3“. M - A/M CO | Fault compresseur 3 „Wie oben, für compresseur Low Lift -pompe Nr.3“. M - A/M CO | Fault compressore 3 „Wie oben, für compressore Low Lift -pompa Nr.3“. M - A/M CO
  134 | Störung Verdichter 4 „Wie oben, für den Verdichter Low Lift -Pumpe Nr.4“. M - A/M CO | Störung Verdichter 4 „Wie oben, für den Verdichter Low Lift -Pumpe Nr.4“. M - A/M CO | Fault compressor 4 „Wie oben, für compressor Low Lift -pump Nr.4“. M - A/M CO | Fault compresseur 4 „Wie oben, für compresseur Low Lift -pompe Nr.4“. M - A/M CO | Fault compressore 4 „Wie oben, für compressore Low Lift -pompa Nr.4“. M - A/M CO
  135 | Störung Verdichter 5 „Wie oben, für den Verdichter Low Lift -Pumpe Nr.5“. M - A/M CO | Störung Verdichter 5 „Wie oben, für den Verdichter Low Lift -Pumpe Nr.5“. M - A/M CO | Fault compressor 5 „Wie oben, für compressor Low Lift -pump Nr.5“. M - A/M CO | Fault compresseur 5 „Wie oben, für compresseur Low Lift -pompe Nr.5“. M - A/M CO | Fault compressore 5 „Wie oben, für compressore Low Lift -pompa Nr.5“. M - A/M CO
  136 | Störung Verdichter 6 „Wie oben, für den Verdichter Low Lift -Pumpe Nr.6“. M - A/M CO | Störung Verdichter 6 „Wie oben, für den Verdichter Low Lift -Pumpe Nr.6“. M - A/M CO | Fault compressor 6 „Wie oben, für compressor Low Lift -pump Nr.6“. M - A/M CO | Fault compresseur 6 „Wie oben, für compresseur Low Lift -pompe Nr.6“. M - A/M CO | Fault compressore 6 „Wie oben, für compressore Low Lift -pompa Nr.6“. M - A/M CO
  137 | Störung Verdichter 7 „Wie oben, für den Verdichter Low Lift -Pumpe Nr.7“. M - A/M CO | Störung Verdichter 7 „Wie oben, für den Verdichter Low Lift -Pumpe Nr.7“. M - A/M CO | Fault compressor 7 „Wie oben, für compressor Low Lift -pump Nr.7“. M - A/M CO | Fault compresseur 7 „Wie oben, für compresseur Low Lift -pompe Nr.7“. M - A/M CO | Fault compressore 7 „Wie oben, für compressore Low Lift -pompa Nr.7“. M - A/M CO
  138 | Störung Verdichter 8 „Wie oben, für den Verdichter Low Lift -Pumpe Nr.8“. M - A/M CO | Störung Verdichter 8 „Wie oben, für den Verdichter Low Lift -Pumpe Nr.8“. M - A/M CO | Fault compressor 8 „Wie oben, für compressor Low Lift -pump Nr.8“. M - A/M CO | Fault compresseur 8 „Wie oben, für compresseur Low Lift -pompe Nr.8“. M - A/M CO | Fault compressore 8 „Wie oben, für compressore Low Lift -pompa Nr.8“. M - A/M CO
  141 | Offline Verdichter 1 | Offline Verdichter 1 | Offline compressor 1 | Offline compresseur 1 | Offline compressore 1
  142 | Offline Verdichter 2 „Wie oben, für den Verdichter Nr.2“. A CO | Offline Verdichter 2 „Wie oben, für den Verdichter Nr.2“. A CO | Offline compressor 2 „Wie oben, für compressor Nr.2“. A CO | Offline compresseur 2 „Wie oben, für compresseur Nr.2“. A CO | Offline compressore 2 „Wie oben, für compressore Nr.2“. A CO
  143 | Offline Verdichter 3 „Wie oben, für den Verdichter Nr.3“. A CO | Offline Verdichter 3 „Wie oben, für den Verdichter Nr.3“. A CO | Offline compressor 3 „Wie oben, für compressor Nr.3“. A CO | Offline compresseur 3 „Wie oben, für compresseur Nr.3“. A CO | Offline compressore 3 „Wie oben, für compressore Nr.3“. A CO
  144 | Offline Verdichter 4 „Wie oben, für den Verdichter Nr.4“. A CO | Offline Verdichter 4 „Wie oben, für den Verdichter Nr.4“. A CO | Offline compressor 4 „Wie oben, für compressor Nr.4“. A CO | Offline compresseur 4 „Wie oben, für compresseur Nr.4“. A CO | Offline compressore 4 „Wie oben, für compressore Nr.4“. A CO
  151 | Wartung Verdichter 1 | Wartung Verdichter 1 | Maintenance compressor 1 | Maintenance compresseur 1 | Maintenance compressore 1
  152 | Wartung Verdichter 2 „Wie oben, für den Verdichter Nr.2“. S - STG0018 | Wartung Verdichter 2 „Wie oben, für den Verdichter Nr.2“. S - STG0018 | Maintenance compressor 2 „Wie oben, für compressor Nr.2“. S - STG0018 | Maintenance compresseur 2 „Wie oben, für compresseur Nr.2“. S - STG0018 | Maintenance compressore 2 „Wie oben, für compressore Nr.2“. S - STG0018
  153 | Wartung Verdichter 3 „Wie oben, für den Verdichter Nr.3“. S - STG0023 | Wartung Verdichter 3 „Wie oben, für den Verdichter Nr.3“. S - STG0023 | Maintenance compressor 3 „Wie oben, für compressor Nr.3“. S - STG0023 | Maintenance compresseur 3 „Wie oben, für compresseur Nr.3“. S - STG0023 | Maintenance compressore 3 „Wie oben, für compressore Nr.3“. S - STG0023
  154 | Wartung Verdichter 4 „Wie oben, für den Verdichter Nr.4“. S - STG0028 | Wartung Verdichter 4 „Wie oben, für den Verdichter Nr.4“. S - STG0028 | Maintenance compressor 4 „Wie oben, für compressor Nr.4“. S - STG0028 | Maintenance compresseur 4 „Wie oben, für compresseur Nr.4“. S - STG0028 | Maintenance compressore 4 „Wie oben, für compressore Nr.4“. S - STG0028
  155 | Wartung Verdichter 5 „Wie oben, für den Verdichter Nr. 5“. S - STG0033 | Wartung Verdichter 5 „Wie oben, für den Verdichter Nr. 5“. S - STG0033 | Maintenance compressor 5 „Wie oben, für compressor Nr. 5“. S - STG0033 | Maintenance compresseur 5 „Wie oben, für compresseur Nr. 5“. S - STG0033 | Maintenance compressore 5 „Wie oben, für compressore Nr. 5“. S - STG0033
  156 | Wartung Verdichter 6 „Wie oben, für den Verdichter Nr. 6“. S - STG0038 | Wartung Verdichter 6 „Wie oben, für den Verdichter Nr. 6“. S - STG0038 | Maintenance compressor 6 „Wie oben, für compressor Nr. 6“. S - STG0038 | Maintenance compresseur 6 „Wie oben, für compresseur Nr. 6“. S - STG0038 | Maintenance compressore 6 „Wie oben, für compressore Nr. 6“. S - STG0038
  157 | Wartung Verdichter 7 „Wie oben, für den Verdichter Nr. 7“. S - STG0043 | Wartung Verdichter 7 „Wie oben, für den Verdichter Nr. 7“. S - STG0043 | Maintenance compressor 7 „Wie oben, für compressor Nr. 7“. S - STG0043 | Maintenance compresseur 7 „Wie oben, für compresseur Nr. 7“. S - STG0043 | Maintenance compressore 7 „Wie oben, für compressore Nr. 7“. S - STG0043
  158 | Wartung Verdichter 8 „Wie oben, für den Verdichter Nr. 8“. S - STG0048 | Wartung Verdichter 8 „Wie oben, für den Verdichter Nr. 8“. S - STG0048 | Maintenance compressor 8 „Wie oben, für compressor Nr. 8“. S - STG0048 | Maintenance compresseur 8 „Wie oben, für compresseur Nr. 8“. S - STG0048 | Maintenance compressore 8 „Wie oben, für compressore Nr. 8“. S - STG0048
  161 | Speisung Motor Verdichter 1 Motor des Verdichters 1 Alarmzustand (nur bei Einheiten mit Turbocor -Verdichtern). A/B CO | Speisung Motor Verdichter 1 Motor des Verdichters 1 Alarmzustand (nur bei Einheiten mit Turbocor -Verdichtern). A/B CO | Speisung motor compressor 1 motor compressors 1 Alarmzustand (nur bei uniten mit Turbocor -compressorn). A/B CO | Speisung moteur compresseur 1 moteur compresseurs 1 Alarmzustand (nur bei unitéen mit Turbocor -compresseurn). A/B CO | Speisung motore compressore 1 motore compressores 1 Alarmzustand (nur bei unitàen mit Turbocor -compressoren). A/B CO
  162 | Speisung Motor Verdichter 2 „Wie oben, für den Verdichter Nr.2“. A/B CO | Speisung Motor Verdichter 2 „Wie oben, für den Verdichter Nr.2“. A/B CO | Speisung motor compressor 2 „Wie oben, für compressor Nr.2“. A/B CO | Speisung moteur compresseur 2 „Wie oben, für compresseur Nr.2“. A/B CO | Speisung motore compressore 2 „Wie oben, für compressore Nr.2“. A/B CO
  163 | Speisung Motor Verdichter 3 „Wie oben, für den Verdichter Nr.3“. A/B CO | Speisung Motor Verdichter 3 „Wie oben, für den Verdichter Nr.3“. A/B CO | Speisung motor compressor 3 „Wie oben, für compressor Nr.3“. A/B CO | Speisung moteur compresseur 3 „Wie oben, für compresseur Nr.3“. A/B CO | Speisung motore compressore 3 „Wie oben, für compressore Nr.3“. A/B CO
  164 | Speisung Motor Verdichter 4 „Wie oben, für den Verdichter Nr.4“. A/B CO | Speisung Motor Verdichter 4 „Wie oben, für den Verdichter Nr.4“. A/B CO | Speisung motor compressor 4 „Wie oben, für compressor Nr.4“. A/B CO | Speisung moteur compresseur 4 „Wie oben, für compresseur Nr.4“. A/B CO | Speisung motore compressore 4 „Wie oben, für compressore Nr.4“. A/B CO
  165 | Speisung Motor Verdichter 5 „Wie oben, für den Verdichter Nr. 5“. A/B CO | Speisung Motor Verdichter 5 „Wie oben, für den Verdichter Nr. 5“. A/B CO | Speisung motor compressor 5 „Wie oben, für compressor Nr. 5“. A/B CO | Speisung moteur compresseur 5 „Wie oben, für compresseur Nr. 5“. A/B CO | Speisung motore compressore 5 „Wie oben, für compressore Nr. 5“. A/B CO
  166 | Speisung Motor Verdichter 6 „Wie oben, für den Verdichter Nr. 6“. A/B CO | Speisung Motor Verdichter 6 „Wie oben, für den Verdichter Nr. 6“. A/B CO | Speisung motor compressor 6 „Wie oben, für compressor Nr. 6“. A/B CO | Speisung moteur compresseur 6 „Wie oben, für compresseur Nr. 6“. A/B CO | Speisung motore compressore 6 „Wie oben, für compressore Nr. 6“. A/B CO
  167 | Speisung Motor Verdichter 7 „Wie oben, für den Verdichter Nr. 7“. A/B CO | Speisung Motor Verdichter 7 „Wie oben, für den Verdichter Nr. 7“. A/B CO | Speisung motor compressor 7 „Wie oben, für compressor Nr. 7“. A/B CO | Speisung moteur compresseur 7 „Wie oben, für compresseur Nr. 7“. A/B CO | Speisung motore compressore 7 „Wie oben, für compressore Nr. 7“. A/B CO
  168 | Speisung Motor Verdichter 8 „Wie oben, für den Verdichter Nr. 8“. A/B CO | Speisung Motor Verdichter 8 „Wie oben, für den Verdichter Nr. 8“. A/B CO | Speisung motor compressor 8 „Wie oben, für compressor Nr. 8“. A/B CO | Speisung moteur compresseur 8 „Wie oben, für compresseur Nr. 8“. A/B CO | Speisung motore compressore 8 „Wie oben, für compressore Nr. 8“. A/B CO
  171 | Timeout Anlauf Verdichter 1 | Timeout Anlauf Verdichter 1 | Start-up timeout compressor 1 | Start-up timeout compresseur 1 | Start-up timeout compressore 1
  172 | Timeout Anlauf Verdichter 2 „Wie oben, für den Verdichter Nr.2“. Turbocor: A/M Schraube: A CO 180s SFT0003 | Timeout Anlauf Verdichter 2 „Wie oben, für den Verdichter Nr.2“. Turbocor: A/M Schraube: A CO 180s SFT0003 | Start-up timeout compressor 2 „Wie oben, für compressor Nr.2“. Turbocor: A/M Schraube: A CO 180s SFT0003 | Start-up timeout compresseur 2 „Wie oben, für compresseur Nr.2“. Turbocor: A/M Schraube: A CO 180s SFT0003 | Start-up timeout compressore 2 „Wie oben, für compressore Nr.2“. Turbocor: A/M Schraube: A CO 180s SFT0003
  173 | Timeout Anlauf Verdichter 3 „Wie oben, für den Verdichter Nr.3“. Turbocor: A/M Schraube: A CO | Timeout Anlauf Verdichter 3 „Wie oben, für den Verdichter Nr.3“. Turbocor: A/M Schraube: A CO | Start-up timeout compressor 3 „Wie oben, für compressor Nr.3“. Turbocor: A/M Schraube: A CO | Start-up timeout compresseur 3 „Wie oben, für compresseur Nr.3“. Turbocor: A/M Schraube: A CO | Start-up timeout compressore 3 „Wie oben, für compressore Nr.3“. Turbocor: A/M Schraube: A CO
  174 | Timeout Anlauf Verdichter 4 „Wie oben, für den Verdichter Nr.4“. Turbocor: A/M CO | Timeout Anlauf Verdichter 4 „Wie oben, für den Verdichter Nr.4“. Turbocor: A/M CO | Start-up timeout compressor 4 „Wie oben, für compressor Nr.4“. Turbocor: A/M CO | Start-up timeout compresseur 4 „Wie oben, für compresseur Nr.4“. Turbocor: A/M CO | Start-up timeout compressore 4 „Wie oben, für compressore Nr.4“. Turbocor: A/M CO
  175 | Timeout Anlauf Verdichter 5 „Wie oben, für den Verdichter Nr. 5“. Turbocor: A/M CO | Timeout Anlauf Verdichter 5 „Wie oben, für den Verdichter Nr. 5“. Turbocor: A/M CO | Start-up timeout compressor 5 „Wie oben, für compressor Nr. 5“. Turbocor: A/M CO | Start-up timeout compresseur 5 „Wie oben, für compresseur Nr. 5“. Turbocor: A/M CO | Start-up timeout compressore 5 „Wie oben, für compressore Nr. 5“. Turbocor: A/M CO
  176 | Timeout Anlauf Verdichter 6 „Wie oben, für den Verdichter Nr. 6“. Turbocor: A/M CO | Timeout Anlauf Verdichter 6 „Wie oben, für den Verdichter Nr. 6“. Turbocor: A/M CO | Start-up timeout compressor 6 „Wie oben, für compressor Nr. 6“. Turbocor: A/M CO | Start-up timeout compresseur 6 „Wie oben, für compresseur Nr. 6“. Turbocor: A/M CO | Start-up timeout compressore 6 „Wie oben, für compressore Nr. 6“. Turbocor: A/M CO
  177 | Timeout Anlauf Verdichter 7 „Wie oben, für den Verdichter Nr. 7“. Turbocor: A/M CO | Timeout Anlauf Verdichter 7 „Wie oben, für den Verdichter Nr. 7“. Turbocor: A/M CO | Start-up timeout compressor 7 „Wie oben, für compressor Nr. 7“. Turbocor: A/M CO | Start-up timeout compresseur 7 „Wie oben, für compresseur Nr. 7“. Turbocor: A/M CO | Start-up timeout compressore 7 „Wie oben, für compressore Nr. 7“. Turbocor: A/M CO
  178 | Timeout Anlauf Verdichter 8 „Wie oben, für den Verdichter Nr. 8“. Turbocor: A/M CO | Timeout Anlauf Verdichter 8 „Wie oben, für den Verdichter Nr. 8“. Turbocor: A/M CO | Start-up timeout compressor 8 „Wie oben, für compressor Nr. 8“. Turbocor: A/M CO | Start-up timeout compresseur 8 „Wie oben, für compresseur Nr. 8“. Turbocor: A/M CO | Start-up timeout compressore 8 „Wie oben, für compressore Nr. 8“. Turbocor: A/M CO
  191 | Economiser Verdichter 1 | Economiser Verdichter 1 | Economiser compressor 1 | Economiser compresseur 1 | Economiser compressore 1
  192 | Economiser Verdichter 2 „Wie oben, für den Verdichter Nr.2“. A CO | Economiser Verdichter 2 „Wie oben, für den Verdichter Nr.2“. A CO | Economiser compressor 2 „Wie oben, für compressor Nr.2“. A CO | Economiser compresseur 2 „Wie oben, für compresseur Nr.2“. A CO | Economiser compressore 2 „Wie oben, für compressore Nr.2“. A CO
  193 | Economiser Verdichter 3 „Wie oben, für den Verdichter Nr.3“. A CO | Economiser Verdichter 3 „Wie oben, für den Verdichter Nr.3“. A CO | Economiser compressor 3 „Wie oben, für compressor Nr.3“. A CO | Economiser compresseur 3 „Wie oben, für compresseur Nr.3“. A CO | Economiser compressore 3 „Wie oben, für compressore Nr.3“. A CO
  194 | Economiser Verdichter 4 „Wie oben, für den Verdichter Nr.4“. A CO | Economiser Verdichter 4 „Wie oben, für den Verdichter Nr.4“. A CO | Economiser compressor 4 „Wie oben, für compressor Nr.4“. A CO | Economiser compresseur 4 „Wie oben, für compresseur Nr.4“. A CO | Economiser compressore 4 „Wie oben, für compressore Nr.4“. A CO
  201 | Störung Kreislauf 1 | Störung Kreislauf 1 | Fault circuit 1 | Fault circuit 1 | Fault circuito 1
  202 | Störung Kreislauf 2 „Wie oben, für den Kreislauf Nr. 2“. S - | Störung Kreislauf 2 „Wie oben, für den Kreislauf Nr. 2“. S - | Fault circuit 2 „Wie oben, für circuit Nr. 2“. S - | Fault circuit 2 „Wie oben, für circuit Nr. 2“. S - | Fault circuito 2 „Wie oben, für circuito Nr. 2“. S -
  203 | Störung Kreislauf 3 „Wie oben, für den Kreislauf Nr. 3“. S - | Störung Kreislauf 3 „Wie oben, für den Kreislauf Nr. 3“. S - | Fault circuit 3 „Wie oben, für circuit Nr. 3“. S - | Fault circuit 3 „Wie oben, für circuit Nr. 3“. S - | Fault circuito 3 „Wie oben, für circuito Nr. 3“. S -
  204 | Störung Kreislauf 4 „Wie oben, für den Kreislauf Nr. 4“. S - | Störung Kreislauf 4 „Wie oben, für den Kreislauf Nr. 4“. S - | Fault circuit 4 „Wie oben, für circuit Nr. 4“. S - | Fault circuit 4 „Wie oben, für circuit Nr. 4“. S - | Fault circuito 4 „Wie oben, für circuito Nr. 4“. S -
  211 | Hochdruck Kreislauf 1 | Hochdruck Kreislauf 1 | Hochdruck circuit 1 | Hochdruck circuit 1 | Hochdruck circuito 1
  212 | Hochdruck Kreislauf 2 „Wie oben, für den Kreislauf Nr. 2“. A/M CI | Hochdruck Kreislauf 2 „Wie oben, für den Kreislauf Nr. 2“. A/M CI | Hochdruck circuit 2 „Wie oben, für circuit Nr. 2“. A/M CI | Hochdruck circuit 2 „Wie oben, für circuit Nr. 2“. A/M CI | Hochdruck circuito 2 „Wie oben, für circuito Nr. 2“. A/M CI
  213 | Hochdruck Kreislauf 3 „Wie oben, für den Kreislauf Nr. 3“. A/M CI | Hochdruck Kreislauf 3 „Wie oben, für den Kreislauf Nr. 3“. A/M CI | Hochdruck circuit 3 „Wie oben, für circuit Nr. 3“. A/M CI | Hochdruck circuit 3 „Wie oben, für circuit Nr. 3“. A/M CI | Hochdruck circuito 3 „Wie oben, für circuito Nr. 3“. A/M CI
  214 | Hochdruck Kreislauf 4 „Wie oben, für den Kreislauf Nr. 4“. A/M CI | Hochdruck Kreislauf 4 „Wie oben, für den Kreislauf Nr. 4“. A/M CI | Hochdruck circuit 4 „Wie oben, für circuit Nr. 4“. A/M CI | Hochdruck circuit 4 „Wie oben, für circuit Nr. 4“. A/M CI | Hochdruck circuito 4 „Wie oben, für circuito Nr. 4“. A/M CI
  221 | Störung Ventilator Kreislauf 1 | Störung Ventilator Kreislauf 1 | Fault fan circuit 1 | Fault ventilateur circuit 1 | Fault ventilatore circuito 1
  222 | Störung Ventilator Kreislauf 2 „Wie oben, für den Kreislauf Nr. 2“. M CI | Störung Ventilator Kreislauf 2 „Wie oben, für den Kreislauf Nr. 2“. M CI | Fault fan circuit 2 „Wie oben, für circuit Nr. 2“. M CI | Fault ventilateur circuit 2 „Wie oben, für circuit Nr. 2“. M CI | Fault ventilatore circuito 2 „Wie oben, für circuito Nr. 2“. M CI
  223 | Störung Ventilator Kreislauf 3 „Wie oben, für den Kreislauf Nr. 3“. M CI | Störung Ventilator Kreislauf 3 „Wie oben, für den Kreislauf Nr. 3“. M CI | Fault fan circuit 3 „Wie oben, für circuit Nr. 3“. M CI | Fault ventilateur circuit 3 „Wie oben, für circuit Nr. 3“. M CI | Fault ventilatore circuito 3 „Wie oben, für circuito Nr. 3“. M CI
  224 | Störung Ventilator Kreislauf 4 „Wie oben, für den Kreislauf Nr. 4“. M CI | Störung Ventilator Kreislauf 4 „Wie oben, für den Kreislauf Nr. 4“. M CI | Fault fan circuit 4 „Wie oben, für circuit Nr. 4“. M CI | Fault ventilateur circuit 4 „Wie oben, für circuit Nr. 4“. M CI | Fault ventilatore circuito 4 „Wie oben, für circuito Nr. 4“. M CI
  231 | Niedriger Druck Kreislauf 1 | Niedriger Druck Kreislauf 1 | Low pressure circuit 1 | Low pressure circuit 1 | Low pressure circuito 1
  232 | Niedriger Druck Kreislauf 2 „Wie oben, für den Kreislauf Nr. 2“. A/M CI | Niedriger Druck Kreislauf 2 „Wie oben, für den Kreislauf Nr. 2“. A/M CI | Low pressure circuit 2 „Wie oben, für circuit Nr. 2“. A/M CI | Low pressure circuit 2 „Wie oben, für circuit Nr. 2“. A/M CI | Low pressure circuito 2 „Wie oben, für circuito Nr. 2“. A/M CI
  233 | Niedriger Druck Kreislauf 3 „Wie oben, für den Kreislauf Nr. 3“. A/M CI | Niedriger Druck Kreislauf 3 „Wie oben, für den Kreislauf Nr. 3“. A/M CI | Low pressure circuit 3 „Wie oben, für circuit Nr. 3“. A/M CI | Low pressure circuit 3 „Wie oben, für circuit Nr. 3“. A/M CI | Low pressure circuito 3 „Wie oben, für circuito Nr. 3“. A/M CI
  234 | Niedriger Druck Kreislauf 4 „Wie oben, für den Kreislauf Nr. 4“. A/M CI | Niedriger Druck Kreislauf 4 „Wie oben, für den Kreislauf Nr. 4“. A/M CI | Low pressure circuit 4 „Wie oben, für circuit Nr. 4“. A/M CI | Low pressure circuit 4 „Wie oben, für circuit Nr. 4“. A/M CI | Low pressure circuito 4 „Wie oben, für circuito Nr. 4“. A/M CI
  241 | Hoher Druck vom Druckmesser 1 | Hoher Druck vom Druckmesser 1 | High pressure vom pressure gauge 1 | High pressure vom manomètre 1 | High pressure vom manometro 1
  242 | Hoher Druck vom Druckmesser 2 „Wie oben, für den Kreislauf Nr. 2“. A/M CI | Hoher Druck vom Druckmesser 2 „Wie oben, für den Kreislauf Nr. 2“. A/M CI | High pressure vom pressure gauge 2 „Wie oben, für circuit Nr. 2“. A/M CI | High pressure vom manomètre 2 „Wie oben, für circuit Nr. 2“. A/M CI | High pressure vom manometro 2 „Wie oben, für circuito Nr. 2“. A/M CI
  243 | Hoher Druck vom Druckmesser 3 „Wie oben, für den Kreislauf Nr. 3“. A/M CI | Hoher Druck vom Druckmesser 3 „Wie oben, für den Kreislauf Nr. 3“. A/M CI | High pressure vom pressure gauge 3 „Wie oben, für circuit Nr. 3“. A/M CI | High pressure vom manomètre 3 „Wie oben, für circuit Nr. 3“. A/M CI | High pressure vom manometro 3 „Wie oben, für circuito Nr. 3“. A/M CI
  244 | Hoher Druck vom Druckmesser 4 „Wie oben, für den Kreislauf Nr. 4“. A/M CI | Hoher Druck vom Druckmesser 4 „Wie oben, für den Kreislauf Nr. 4“. A/M CI | High pressure vom pressure gauge 4 „Wie oben, für circuit Nr. 4“. A/M CI | High pressure vom manomètre 4 „Wie oben, für circuit Nr. 4“. A/M CI | High pressure vom manometro 4 „Wie oben, für circuito Nr. 4“. A/M CI
  251 | Timeout Anlauf Kreislauf 1 Möglicher Anlaufversuch bei Freon -Mangel im Kreislauf Nr. 1. A CI SFT0003 | Timeout Anlauf Kreislauf 1 Möglicher Anlaufversuch bei Freon -Mangel im Kreislauf Nr. 1. A CI SFT0003 | Start-up timeout circuit 1 Möglicher Anlaufversuch bei Freon -Mangel im circuit Nr. 1. A CI SFT0003 | Start-up timeout circuit 1 Möglicher Anlaufversuch bei Freon -Mangel im circuit Nr. 1. A CI SFT0003 | Start-up timeout circuito 1 Möglicher Anlaufversuch bei Freon -Mangel im circuito Nr. 1. A CI SFT0003
  252 | Timeout Anlauf Kreislauf 2 „Wie oben, für den Kreislauf Nr. 2“. A CI | Timeout Anlauf Kreislauf 2 „Wie oben, für den Kreislauf Nr. 2“. A CI | Start-up timeout circuit 2 „Wie oben, für circuit Nr. 2“. A CI | Start-up timeout circuit 2 „Wie oben, für circuit Nr. 2“. A CI | Start-up timeout circuito 2 „Wie oben, für circuito Nr. 2“. A CI
  253 | Timeout Anlauf Kreislauf 3 „Wie oben, für den Kreislauf Nr. 3“. A CI | Timeout Anlauf Kreislauf 3 „Wie oben, für den Kreislauf Nr. 3“. A CI | Start-up timeout circuit 3 „Wie oben, für circuit Nr. 3“. A CI | Start-up timeout circuit 3 „Wie oben, für circuit Nr. 3“. A CI | Start-up timeout circuito 3 „Wie oben, für circuito Nr. 3“. A CI
  254 | Timeout Anlauf Kreislauf 4 „Wie oben, für den Kreislauf Nr. 4“. A CI | Timeout Anlauf Kreislauf 4 „Wie oben, für den Kreislauf Nr. 4“. A CI | Start-up timeout circuit 4 „Wie oben, für circuit Nr. 4“. A CI | Start-up timeout circuit 4 „Wie oben, für circuit Nr. 4“. A CI | Start-up timeout circuito 4 „Wie oben, für circuito Nr. 4“. A CI
  261 | Kein Freon Kreislauf 1 | Kein Freon Kreislauf 1 | No refrigerant circuit 1 | No refrigerant circuit 1 | No refrigerant circuito 1
  262 | Kein Freon Kreislauf 2 „Wie oben, für den Kreislauf Nr. 2“. A CI | Kein Freon Kreislauf 2 „Wie oben, für den Kreislauf Nr. 2“. A CI | No refrigerant circuit 2 „Wie oben, für circuit Nr. 2“. A CI | No refrigerant circuit 2 „Wie oben, für circuit Nr. 2“. A CI | No refrigerant circuito 2 „Wie oben, für circuito Nr. 2“. A CI
  263 | Kein Freon Kreislauf 3 „Wie oben, für den Kreislauf Nr. 3“. A CI | Kein Freon Kreislauf 3 „Wie oben, für den Kreislauf Nr. 3“. A CI | No refrigerant circuit 3 „Wie oben, für circuit Nr. 3“. A CI | No refrigerant circuit 3 „Wie oben, für circuit Nr. 3“. A CI | No refrigerant circuito 3 „Wie oben, für circuito Nr. 3“. A CI
  264 | Kein Freon Kreislauf 4 „Wie oben, für den Kreislauf Nr. 4“. A CI | Kein Freon Kreislauf 4 „Wie oben, für den Kreislauf Nr. 4“. A CI | No refrigerant circuit 4 „Wie oben, für circuit Nr. 4“. A CI | No refrigerant circuit 4 „Wie oben, für circuit Nr. 4“. A CI | No refrigerant circuito 4 „Wie oben, für circuito Nr. 4“. A CI
  271 | Lamellenregister Kreislauf 1 | Lamellenregister Kreislauf 1 | coil circuit 1 | batterie à ailettes circuit 1 | batteria alettata circuito 1
  272 | Lamellenregister Kreislauf 2 „Wie oben, für den Kreislauf Nr. 2“. S-M CI | Lamellenregister Kreislauf 2 „Wie oben, für den Kreislauf Nr. 2“. S-M CI | coil circuit 2 „Wie oben, für circuit Nr. 2“. S-M CI | batterie à ailettes circuit 2 „Wie oben, für circuit Nr. 2“. S-M CI | batteria alettata circuito 2 „Wie oben, für circuito Nr. 2“. S-M CI
  273 | Lamellenregister Kreislauf 3 „Wie oben, für den Kreislauf Nr. 3“. S-M CI | Lamellenregister Kreislauf 3 „Wie oben, für den Kreislauf Nr. 3“. S-M CI | coil circuit 3 „Wie oben, für circuit Nr. 3“. S-M CI | batterie à ailettes circuit 3 „Wie oben, für circuit Nr. 3“. S-M CI | batteria alettata circuito 3 „Wie oben, für circuito Nr. 3“. S-M CI
  274 | Lamellenregister Kreislauf 4 „Wie oben, für den Kreislauf Nr. 4“. S-M CI | Lamellenregister Kreislauf 4 „Wie oben, für den Kreislauf Nr. 4“. S-M CI | coil circuit 4 „Wie oben, für circuit Nr. 4“. S-M CI | batterie à ailettes circuit 4 „Wie oben, für circuit Nr. 4“. S-M CI | batteria alettata circuito 4 „Wie oben, für circuito Nr. 4“. S-M CI
  281 | Verdampfungsdruck zu niedrig Kreislauf Nr. 1 Möglicherweise ist kein Freon im Kreislauf Nr. 1, da er mit einem Verdampfungsdruck arbeitet, der unter dem eingestellten Grenzwert liegt. M CI STG0068 STG0167 STG0168 | Verdampfungsdruck zu niedrig Kreislauf Nr. 1 Möglicherweise ist kein Freon im Kreislauf Nr. 1, da er mit einem Verdampfungsdruck arbeitet, der unter dem eingestellten Grenzwert liegt. M CI STG0068 STG0167 STG0168 | Verdampfungsdruck zu niedrig circuit Nr. 1 Möglicherweise ist kein Freon im circuit Nr. 1, da er mit einem Verdampfungsdruck arbeitet, unter eingestellten Grenzwert liegt. M CI STG0068 STG0167 STG0168 | Verdampfungsdruck zu niedrig circuit Nr. 1 Möglicherweise ist kein Freon im circuit Nr. 1, da er mit einem Verdampfungsdruck arbeitet, unter eingestellten Grenzwert liegt. M CI STG0068 STG0167 STG0168 | Verdampfungsdruck zu niedrig circuito Nr. 1 Möglicherweise ist kein Freon im circuito Nr. 1, da er mit einem Verdampfungsdruck arbeitet, unter eingestellten Grenzwert liegt. M CI STG0068 STG0167 STG0168
  282 | Verdampfungsdruck zu niedrig Kreislauf Nr. 2 „Wie oben, für den Kreislauf Nr. 2“. M CI | Verdampfungsdruck zu niedrig Kreislauf Nr. 2 „Wie oben, für den Kreislauf Nr. 2“. M CI | Verdampfungsdruck zu niedrig circuit Nr. 2 „Wie oben, für circuit Nr. 2“. M CI | Verdampfungsdruck zu niedrig circuit Nr. 2 „Wie oben, für circuit Nr. 2“. M CI | Verdampfungsdruck zu niedrig circuito Nr. 2 „Wie oben, für circuito Nr. 2“. M CI
  283 | Verdampfungsdruck zu niedrig Kreislauf Nr. 3 „Wie oben, für den Kreislauf Nr. 3“. M CI | Verdampfungsdruck zu niedrig Kreislauf Nr. 3 „Wie oben, für den Kreislauf Nr. 3“. M CI | Verdampfungsdruck zu niedrig circuit Nr. 3 „Wie oben, für circuit Nr. 3“. M CI | Verdampfungsdruck zu niedrig circuit Nr. 3 „Wie oben, für circuit Nr. 3“. M CI | Verdampfungsdruck zu niedrig circuito Nr. 3 „Wie oben, für circuito Nr. 3“. M CI
  284 | Verdampfungsdruck zu niedrig Kreislauf Nr. 4 „Wie oben, für den Kreislauf Nr. 4“. M CI | Verdampfungsdruck zu niedrig Kreislauf Nr. 4 „Wie oben, für den Kreislauf Nr. 4“. M CI | Verdampfungsdruck zu niedrig circuit Nr. 4 „Wie oben, für circuit Nr. 4“. M CI | Verdampfungsdruck zu niedrig circuit Nr. 4 „Wie oben, für circuit Nr. 4“. M CI | Verdampfungsdruck zu niedrig circuito Nr. 4 „Wie oben, für circuito Nr. 4“. M CI
  291 | Zu wenig Freon im Kreislauf Nr. 1 Das Freon im Kreislauf Nr. 1 ist nicht ausreichend, da die Einheit unter der Approach -Grenze gearbeitet hat. A/M CI SFT0022 | Zu wenig Freon im Kreislauf Nr. 1 Das Freon im Kreislauf Nr. 1 ist nicht ausreichend, da die Einheit unter der Approach -Grenze gearbeitet hat. A/M CI SFT0022 | Zu wenig Freon im circuit Nr. 1 Freon im circuit Nr. 1 ist nicht ausreichend, da unit unter Approach -Grenze gearbeitet hat. A/M CI SFT0022 | Zu wenig Freon im circuit Nr. 1 Freon im circuit Nr. 1 ist nicht ausreichend, da unité unter Approach -Grenze gearbeitet hat. A/M CI SFT0022 | Zu wenig Freon im circuito Nr. 1 Freon im circuito Nr. 1 ist nicht ausreichend, da unità unter Approach -Grenze gearbeitet hat. A/M CI SFT0022
  292 | Zu wenig Freon im Kreislauf Nr. 2 „Wie oben, für den Kreislauf Nr. 2“. A/M CI | Zu wenig Freon im Kreislauf Nr. 2 „Wie oben, für den Kreislauf Nr. 2“. A/M CI | Zu wenig Freon im circuit Nr. 2 „Wie oben, für circuit Nr. 2“. A/M CI | Zu wenig Freon im circuit Nr. 2 „Wie oben, für circuit Nr. 2“. A/M CI | Zu wenig Freon im circuito Nr. 2 „Wie oben, für circuito Nr. 2“. A/M CI
  293 | Zu wenig Freon im Kreislauf Nr. 3 „Wie oben, für den Kreislauf Nr. 3“. A/M CI | Zu wenig Freon im Kreislauf Nr. 3 „Wie oben, für den Kreislauf Nr. 3“. A/M CI | Zu wenig Freon im circuit Nr. 3 „Wie oben, für circuit Nr. 3“. A/M CI | Zu wenig Freon im circuit Nr. 3 „Wie oben, für circuit Nr. 3“. A/M CI | Zu wenig Freon im circuito Nr. 3 „Wie oben, für circuito Nr. 3“. A/M CI
  294 | Zu wenig Freon im Kreislauf Nr. 4 „Wie oben, für den Kreislauf Nr. 4“. A/M CI | Zu wenig Freon im Kreislauf Nr. 4 „Wie oben, für den Kreislauf Nr. 4“. A/M CI | Zu wenig Freon im circuit Nr. 4 „Wie oben, für circuit Nr. 4“. A/M CI | Zu wenig Freon im circuit Nr. 4 „Wie oben, für circuit Nr. 4“. A/M CI | Zu wenig Freon im circuito Nr. 4 „Wie oben, für circuito Nr. 4“. A/M CI
  301 | Temperatur Inverter Verdichter 1 Übertemperatur am Inverter des Verdichters Nr.1 (nur bei Einheiten mit Turbocor -Verdichtern). A/M/B CO | Temperatur Inverter Verdichter 1 Übertemperatur am Inverter des Verdichters Nr.1 (nur bei Einheiten mit Turbocor -Verdichtern). A/M/B CO | Temperatur inverter compressor 1 Übertemperatur am inverter compressors Nr.1 (nur bei uniten mit Turbocor -compressorn). A/M/B CO | Temperatur variateur compresseur 1 Übertemperatur am variateur compresseurs Nr.1 (nur bei unitéen mit Turbocor -compresseurn). A/M/B CO | Temperatur inverter compressore 1 Übertemperatur am inverter compressores Nr.1 (nur bei unitàen mit Turbocor -compressoren). A/M/B CO
  302 | Temperatur Inverter Verdichter 2 „Wie oben, für den Verdichter Nr.2“. A/M/B CO | Temperatur Inverter Verdichter 2 „Wie oben, für den Verdichter Nr.2“. A/M/B CO | Temperatur inverter compressor 2 „Wie oben, für compressor Nr.2“. A/M/B CO | Temperatur variateur compresseur 2 „Wie oben, für compresseur Nr.2“. A/M/B CO | Temperatur inverter compressore 2 „Wie oben, für compressore Nr.2“. A/M/B CO
  303 | Temperatur Inverter Verdichter 3 „Wie oben, für den Verdichter Nr.3“. A/M/B CO | Temperatur Inverter Verdichter 3 „Wie oben, für den Verdichter Nr.3“. A/M/B CO | Temperatur inverter compressor 3 „Wie oben, für compressor Nr.3“. A/M/B CO | Temperatur variateur compresseur 3 „Wie oben, für compresseur Nr.3“. A/M/B CO | Temperatur inverter compressore 3 „Wie oben, für compressore Nr.3“. A/M/B CO
  304 | Temperatur Inverter Verdichter 4 „Wie oben, für den Verdichter Nr.4“. A/M/B CO | Temperatur Inverter Verdichter 4 „Wie oben, für den Verdichter Nr.4“. A/M/B CO | Temperatur inverter compressor 4 „Wie oben, für compressor Nr.4“. A/M/B CO | Temperatur variateur compresseur 4 „Wie oben, für compresseur Nr.4“. A/M/B CO | Temperatur inverter compressore 4 „Wie oben, für compressore Nr.4“. A/M/B CO
  305 | Temperatur Inverter Verdichter 5 „Wie oben, für den Verdichter Nr. 5“. A/M/B CO | Temperatur Inverter Verdichter 5 „Wie oben, für den Verdichter Nr. 5“. A/M/B CO | Temperatur inverter compressor 5 „Wie oben, für compressor Nr. 5“. A/M/B CO | Temperatur variateur compresseur 5 „Wie oben, für compresseur Nr. 5“. A/M/B CO | Temperatur inverter compressore 5 „Wie oben, für compressore Nr. 5“. A/M/B CO
  306 | Temperatur Inverter Verdichter 6 „Wie oben, für den Verdichter Nr. 6“. A/M/B CO | Temperatur Inverter Verdichter 6 „Wie oben, für den Verdichter Nr. 6“. A/M/B CO | Temperatur inverter compressor 6 „Wie oben, für compressor Nr. 6“. A/M/B CO | Temperatur variateur compresseur 6 „Wie oben, für compresseur Nr. 6“. A/M/B CO | Temperatur inverter compressore 6 „Wie oben, für compressore Nr. 6“. A/M/B CO
  307 | Temperatur Inverter Verdichter 7 „Wie oben, für den Verdichter Nr. 7“. A/M/B CO | Temperatur Inverter Verdichter 7 „Wie oben, für den Verdichter Nr. 7“. A/M/B CO | Temperatur inverter compressor 7 „Wie oben, für compressor Nr. 7“. A/M/B CO | Temperatur variateur compresseur 7 „Wie oben, für compresseur Nr. 7“. A/M/B CO | Temperatur inverter compressore 7 „Wie oben, für compressore Nr. 7“. A/M/B CO
  308 | Temperatur Inverter Verdichter 8 „Wie oben, für den Verdichter Nr. 8“. A/M/B CO | Temperatur Inverter Verdichter 8 „Wie oben, für den Verdichter Nr. 8“. A/M/B CO | Temperatur inverter compressor 8 „Wie oben, für compressor Nr. 8“. A/M/B CO | Temperatur variateur compresseur 8 „Wie oben, für compresseur Nr. 8“. A/M/B CO | Temperatur inverter compressore 8 „Wie oben, für compressore Nr. 8“. A/M/B CO
  311 | Austrittstemperatur Verdichter 1 Übertemperatur am Auslass des Verdichters Nr.1 (nur bei Einheiten mit Turbocor -Verdichtern). A/M/B CO | Austrittstemperatur Verdichter 1 Übertemperatur am Auslass des Verdichters Nr.1 (nur bei Einheiten mit Turbocor -Verdichtern). A/M/B CO | Discharge temperature compressor 1 Übertemperatur am Auslass compressors Nr.1 (nur bei uniten mit Turbocor -compressorn). A/M/B CO | Discharge temperature compresseur 1 Übertemperatur am Auslass compresseurs Nr.1 (nur bei unitéen mit Turbocor -compresseurn). A/M/B CO | Discharge temperature compressore 1 Übertemperatur am Auslass compressores Nr.1 (nur bei unitàen mit Turbocor -compressoren). A/M/B CO
  312 | Austrittstemperatur Verdichter 2 „Wie oben, für den Verdichter Nr.2“. A/M/B CO | Austrittstemperatur Verdichter 2 „Wie oben, für den Verdichter Nr.2“. A/M/B CO | Discharge temperature compressor 2 „Wie oben, für compressor Nr.2“. A/M/B CO | Discharge temperature compresseur 2 „Wie oben, für compresseur Nr.2“. A/M/B CO | Discharge temperature compressore 2 „Wie oben, für compressore Nr.2“. A/M/B CO
  313 | Austrittstemperatur Verdichter 3 „Wie oben, für den Verdichter Nr.3“. A/M/B CO | Austrittstemperatur Verdichter 3 „Wie oben, für den Verdichter Nr.3“. A/M/B CO | Discharge temperature compressor 3 „Wie oben, für compressor Nr.3“. A/M/B CO | Discharge temperature compresseur 3 „Wie oben, für compresseur Nr.3“. A/M/B CO | Discharge temperature compressore 3 „Wie oben, für compressore Nr.3“. A/M/B CO
  314 | Austrittstemperatur Verdichter 4 „Wie oben, für den Verdichter Nr.4“. A/M/B CO | Austrittstemperatur Verdichter 4 „Wie oben, für den Verdichter Nr.4“. A/M/B CO | Discharge temperature compressor 4 „Wie oben, für compressor Nr.4“. A/M/B CO | Discharge temperature compresseur 4 „Wie oben, für compresseur Nr.4“. A/M/B CO | Discharge temperature compressore 4 „Wie oben, für compressore Nr.4“. A/M/B CO
  315 | Austrittstemperatur Verdichter 5 „Wie oben, für den Verdichter Nr. 5“. A/M/B CO | Austrittstemperatur Verdichter 5 „Wie oben, für den Verdichter Nr. 5“. A/M/B CO | Discharge temperature compressor 5 „Wie oben, für compressor Nr. 5“. A/M/B CO | Discharge temperature compresseur 5 „Wie oben, für compresseur Nr. 5“. A/M/B CO | Discharge temperature compressore 5 „Wie oben, für compressore Nr. 5“. A/M/B CO
  316 | Austrittstemperatur Verdichter 6 „Wie oben, für den Verdichter Nr. 6“. A/M/B CO | Austrittstemperatur Verdichter 6 „Wie oben, für den Verdichter Nr. 6“. A/M/B CO | Discharge temperature compressor 6 „Wie oben, für compressor Nr. 6“. A/M/B CO | Discharge temperature compresseur 6 „Wie oben, für compresseur Nr. 6“. A/M/B CO | Discharge temperature compressore 6 „Wie oben, für compressore Nr. 6“. A/M/B CO
  317 | Austrittstemperatur Verdichter 7 „Wie oben, für den Verdichter Nr. 7“. A/M/B CO | Austrittstemperatur Verdichter 7 „Wie oben, für den Verdichter Nr. 7“. A/M/B CO | Discharge temperature compressor 7 „Wie oben, für compressor Nr. 7“. A/M/B CO | Discharge temperature compresseur 7 „Wie oben, für compresseur Nr. 7“. A/M/B CO | Discharge temperature compressore 7 „Wie oben, für compressore Nr. 7“. A/M/B CO
  318 | Austrittstemperatur Verdichter 8 „Wie oben, für den Verdichter Nr. 8“. A/M/B CO | Austrittstemperatur Verdichter 8 „Wie oben, für den Verdichter Nr. 8“. A/M/B CO | Discharge temperature compressor 8 „Wie oben, für compressor Nr. 8“. A/M/B CO | Discharge temperature compresseur 8 „Wie oben, für compresseur Nr. 8“. A/M/B CO | Discharge temperature compressore 8 „Wie oben, für compressore Nr. 8“. A/M/B CO
  321 | Niedriger Druck Verdichter 1 | Niedriger Druck Verdichter 1 | Low pressure compressor 1 | Low pressure compresseur 1 | Low pressure compressore 1
  322 | Niedriger Druck Verdichter 2 „Wie oben, für den Verdichter Nr.2“. Turbocor: A/M/B Schraube: A/M CO | Niedriger Druck Verdichter 2 „Wie oben, für den Verdichter Nr.2“. Turbocor: A/M/B Schraube: A/M CO | Low pressure compressor 2 „Wie oben, für compressor Nr.2“. Turbocor: A/M/B Schraube: A/M CO | Low pressure compresseur 2 „Wie oben, für compresseur Nr.2“. Turbocor: A/M/B Schraube: A/M CO | Low pressure compressore 2 „Wie oben, für compressore Nr.2“. Turbocor: A/M/B Schraube: A/M CO
  323 | Niedriger Druck Verdichter 3 „Wie oben, für den Verdichter Nr.3“. Turbocor: A/M/B Schraube: A/M CO | Niedriger Druck Verdichter 3 „Wie oben, für den Verdichter Nr.3“. Turbocor: A/M/B Schraube: A/M CO | Low pressure compressor 3 „Wie oben, für compressor Nr.3“. Turbocor: A/M/B Schraube: A/M CO | Low pressure compresseur 3 „Wie oben, für compresseur Nr.3“. Turbocor: A/M/B Schraube: A/M CO | Low pressure compressore 3 „Wie oben, für compressore Nr.3“. Turbocor: A/M/B Schraube: A/M CO
  324 | Niedriger Druck Verdichter 4 „Wie oben, für den Verdichter Nr.4“. Turbocor: A/M/B Schraube: A/M CO | Niedriger Druck Verdichter 4 „Wie oben, für den Verdichter Nr.4“. Turbocor: A/M/B Schraube: A/M CO | Low pressure compressor 4 „Wie oben, für compressor Nr.4“. Turbocor: A/M/B Schraube: A/M CO | Low pressure compresseur 4 „Wie oben, für compresseur Nr.4“. Turbocor: A/M/B Schraube: A/M CO | Low pressure compressore 4 „Wie oben, für compressore Nr.4“. Turbocor: A/M/B Schraube: A/M CO
  325 | Niedriger Druck Verdichter 5 „Wie oben, für den Verdichter Nr. 5“. Turbocor: A/M/B Schraube: A/M CO | Niedriger Druck Verdichter 5 „Wie oben, für den Verdichter Nr. 5“. Turbocor: A/M/B Schraube: A/M CO | Low pressure compressor 5 „Wie oben, für compressor Nr. 5“. Turbocor: A/M/B Schraube: A/M CO | Low pressure compresseur 5 „Wie oben, für compresseur Nr. 5“. Turbocor: A/M/B Schraube: A/M CO | Low pressure compressore 5 „Wie oben, für compressore Nr. 5“. Turbocor: A/M/B Schraube: A/M CO
  326 | Niedriger Druck Verdichter 6 „Wie oben, für den Verdichter Nr. 6“. Turbocor: A/M/B Schraube: A/M CO | Niedriger Druck Verdichter 6 „Wie oben, für den Verdichter Nr. 6“. Turbocor: A/M/B Schraube: A/M CO | Low pressure compressor 6 „Wie oben, für compressor Nr. 6“. Turbocor: A/M/B Schraube: A/M CO | Low pressure compresseur 6 „Wie oben, für compresseur Nr. 6“. Turbocor: A/M/B Schraube: A/M CO | Low pressure compressore 6 „Wie oben, für compressore Nr. 6“. Turbocor: A/M/B Schraube: A/M CO
  327 | Niedriger Druck Verdichter 7 „Wie oben, für den Verdichter Nr. 7“. Turbocor: A/M/B Schraube: A/M CO | Niedriger Druck Verdichter 7 „Wie oben, für den Verdichter Nr. 7“. Turbocor: A/M/B Schraube: A/M CO | Low pressure compressor 7 „Wie oben, für compressor Nr. 7“. Turbocor: A/M/B Schraube: A/M CO | Low pressure compresseur 7 „Wie oben, für compresseur Nr. 7“. Turbocor: A/M/B Schraube: A/M CO | Low pressure compressore 7 „Wie oben, für compressore Nr. 7“. Turbocor: A/M/B Schraube: A/M CO
  328 | Niedriger Druck Verdichter 8 „Wie oben, für den Verdichter Nr. 8“. Turbocor: A/M/B Schraube: A/M CO | Niedriger Druck Verdichter 8 „Wie oben, für den Verdichter Nr. 8“. Turbocor: A/M/B Schraube: A/M CO | Low pressure compressor 8 „Wie oben, für compressor Nr. 8“. Turbocor: A/M/B Schraube: A/M CO | Low pressure compresseur 8 „Wie oben, für compresseur Nr. 8“. Turbocor: A/M/B Schraube: A/M CO | Low pressure compressore 8 „Wie oben, für compressore Nr. 8“. Turbocor: A/M/B Schraube: A/M CO
  331 | Hoher Druck Verdichter 1 | Hoher Druck Verdichter 1 | High pressure compressor 1 | High pressure compresseur 1 | High pressure compressore 1
  332 | Hoher Druck Verdichter 2 „Wie oben, für den Verdichter Nr.2“. Turbocor: A/M/B Schraube: A/M CO | Hoher Druck Verdichter 2 „Wie oben, für den Verdichter Nr.2“. Turbocor: A/M/B Schraube: A/M CO | High pressure compressor 2 „Wie oben, für compressor Nr.2“. Turbocor: A/M/B Schraube: A/M CO | High pressure compresseur 2 „Wie oben, für compresseur Nr.2“. Turbocor: A/M/B Schraube: A/M CO | High pressure compressore 2 „Wie oben, für compressore Nr.2“. Turbocor: A/M/B Schraube: A/M CO
  333 | Hoher Druck Verdichter 3 „Wie oben, für den Verdichter Nr.3“. Turbocor: A/M/B Schraube: A/M CO | Hoher Druck Verdichter 3 „Wie oben, für den Verdichter Nr.3“. Turbocor: A/M/B Schraube: A/M CO | High pressure compressor 3 „Wie oben, für compressor Nr.3“. Turbocor: A/M/B Schraube: A/M CO | High pressure compresseur 3 „Wie oben, für compresseur Nr.3“. Turbocor: A/M/B Schraube: A/M CO | High pressure compressore 3 „Wie oben, für compressore Nr.3“. Turbocor: A/M/B Schraube: A/M CO
  334 | Hoher Druck Verdichter 4 „Wie oben, für den Verdichter Nr.4“. Turbocor: A/M/B Schraube: A/M CO | Hoher Druck Verdichter 4 „Wie oben, für den Verdichter Nr.4“. Turbocor: A/M/B Schraube: A/M CO | High pressure compressor 4 „Wie oben, für compressor Nr.4“. Turbocor: A/M/B Schraube: A/M CO | High pressure compresseur 4 „Wie oben, für compresseur Nr.4“. Turbocor: A/M/B Schraube: A/M CO | High pressure compressore 4 „Wie oben, für compressore Nr.4“. Turbocor: A/M/B Schraube: A/M CO
  335 | Hoher Druck Verdichter 5 „Wie oben, für den Verdichter Nr. 5“. Turbocor: A/M/B CO | Hoher Druck Verdichter 5 „Wie oben, für den Verdichter Nr. 5“. Turbocor: A/M/B CO | High pressure compressor 5 „Wie oben, für compressor Nr. 5“. Turbocor: A/M/B CO | High pressure compresseur 5 „Wie oben, für compresseur Nr. 5“. Turbocor: A/M/B CO | High pressure compressore 5 „Wie oben, für compressore Nr. 5“. Turbocor: A/M/B CO
  336 | Hoher Druck Verdichter 6 „Wie oben, für den Verdichter Nr. 6“. Turbocor: A/M/B CO | Hoher Druck Verdichter 6 „Wie oben, für den Verdichter Nr. 6“. Turbocor: A/M/B CO | High pressure compressor 6 „Wie oben, für compressor Nr. 6“. Turbocor: A/M/B CO | High pressure compresseur 6 „Wie oben, für compresseur Nr. 6“. Turbocor: A/M/B CO | High pressure compressore 6 „Wie oben, für compressore Nr. 6“. Turbocor: A/M/B CO
  337 | Hoher Druck Verdichter 7 „Wie oben, für den Verdichter Nr. 7“. Turbocor: A/M/B CO | Hoher Druck Verdichter 7 „Wie oben, für den Verdichter Nr. 7“. Turbocor: A/M/B CO | High pressure compressor 7 „Wie oben, für compressor Nr. 7“. Turbocor: A/M/B CO | High pressure compresseur 7 „Wie oben, für compresseur Nr. 7“. Turbocor: A/M/B CO | High pressure compressore 7 „Wie oben, für compressore Nr. 7“. Turbocor: A/M/B CO
  338 | Hoher Druck Verdichter 8 „Wie oben, für den Verdichter Nr. 8“. Turbocor: A/M/B CO | Hoher Druck Verdichter 8 „Wie oben, für den Verdichter Nr. 8“. Turbocor: A/M/B CO | High pressure compressor 8 „Wie oben, für compressor Nr. 8“. Turbocor: A/M/B CO | High pressure compresseur 8 „Wie oben, für compresseur Nr. 8“. Turbocor: A/M/B CO | High pressure compressore 8 „Wie oben, für compressore Nr. 8“. Turbocor: A/M/B CO
  341 | Stromaufnahme Verdichter 1 Stromaufnahme des Verdichters Nr.1 liegt über dem zulässigen Höchstwert (nur bei Einheiten mit Turbocor -Verdichtern). A/M/B CO | Stromaufnahme Verdichter 1 Stromaufnahme des Verdichters Nr.1 liegt über dem zulässigen Höchstwert (nur bei Einheiten mit Turbocor -Verdichtern). A/M/B CO | Current draw compressor 1 Stromaufnahme compressors Nr.1 liegt über zulässigen Höchstwert (nur bei uniten mit Turbocor -compressorn). A/M/B CO | Current draw compresseur 1 Stromaufnahme compresseurs Nr.1 liegt über zulässigen Höchstwert (nur bei unitéen mit Turbocor -compresseurn). A/M/B CO | Current draw compressore 1 Stromaufnahme compressores Nr.1 liegt über zulässigen Höchstwert (nur bei unitàen mit Turbocor -compressoren). A/M/B CO
  342 | Stromaufnahme Verdichter 2 „Wie oben, für den Verdichter Nr.2“. A/M/B CO | Stromaufnahme Verdichter 2 „Wie oben, für den Verdichter Nr.2“. A/M/B CO | Current draw compressor 2 „Wie oben, für compressor Nr.2“. A/M/B CO | Current draw compresseur 2 „Wie oben, für compresseur Nr.2“. A/M/B CO | Current draw compressore 2 „Wie oben, für compressore Nr.2“. A/M/B CO
  343 | Stromaufnahme Verdichter 3 „Wie oben, für den Verdichter Nr.3“. A/M/B CO | Stromaufnahme Verdichter 3 „Wie oben, für den Verdichter Nr.3“. A/M/B CO | Current draw compressor 3 „Wie oben, für compressor Nr.3“. A/M/B CO | Current draw compresseur 3 „Wie oben, für compresseur Nr.3“. A/M/B CO | Current draw compressore 3 „Wie oben, für compressore Nr.3“. A/M/B CO
  344 | Stromaufnahme Verdichter 4 „Wie oben, für den Verdichter Nr.4“. A/M/B CO | Stromaufnahme Verdichter 4 „Wie oben, für den Verdichter Nr.4“. A/M/B CO | Current draw compressor 4 „Wie oben, für compressor Nr.4“. A/M/B CO | Current draw compresseur 4 „Wie oben, für compresseur Nr.4“. A/M/B CO | Current draw compressore 4 „Wie oben, für compressore Nr.4“. A/M/B CO
  345 | Stromaufnahme Verdichter 5 „Wie oben, für den Verdichter Nr.4“. A/M/B CO | Stromaufnahme Verdichter 5 „Wie oben, für den Verdichter Nr.4“. A/M/B CO | Current draw compressor 5 „Wie oben, für compressor Nr.4“. A/M/B CO | Current draw compresseur 5 „Wie oben, für compresseur Nr.4“. A/M/B CO | Current draw compressore 5 „Wie oben, für compressore Nr.4“. A/M/B CO
  346 | Stromaufnahme Verdichter 6 „Wie oben, für den Verdichter Nr.4“. A/M/B CO | Stromaufnahme Verdichter 6 „Wie oben, für den Verdichter Nr.4“. A/M/B CO | Current draw compressor 6 „Wie oben, für compressor Nr.4“. A/M/B CO | Current draw compresseur 6 „Wie oben, für compresseur Nr.4“. A/M/B CO | Current draw compressore 6 „Wie oben, für compressore Nr.4“. A/M/B CO
  347 | Stromaufnahme Verdichter 7 „Wie oben, für den Verdichter Nr.4“. A/M/B CO | Stromaufnahme Verdichter 7 „Wie oben, für den Verdichter Nr.4“. A/M/B CO | Current draw compressor 7 „Wie oben, für compressor Nr.4“. A/M/B CO | Current draw compresseur 7 „Wie oben, für compresseur Nr.4“. A/M/B CO | Current draw compressore 7 „Wie oben, für compressore Nr.4“. A/M/B CO
  348 | Stromaufnahme Verdichter 8 „Wie oben, für den Verdichter Nr.4“. A/M/B CO | Stromaufnahme Verdichter 8 „Wie oben, für den Verdichter Nr.4“. A/M/B CO | Current draw compressor 8 „Wie oben, für compressor Nr.4“. A/M/B CO | Current draw compresseur 8 „Wie oben, für compresseur Nr.4“. A/M/B CO | Current draw compressore 8 „Wie oben, für compressore Nr.4“. A/M/B CO
  351 | Rotortemperatur Verdichter 1 | Rotortemperatur Verdichter 1 | Rotor temperature compressor 1 | Rotor temperature compresseur 1 | Rotor temperature compressore 1
  352 | Rotortemperatur Verdichter 2 „Wie oben, für den Verdichter Nr.2“. A/M/B CO | Rotortemperatur Verdichter 2 „Wie oben, für den Verdichter Nr.2“. A/M/B CO | Rotor temperature compressor 2 „Wie oben, für compressor Nr.2“. A/M/B CO | Rotor temperature compresseur 2 „Wie oben, für compresseur Nr.2“. A/M/B CO | Rotor temperature compressore 2 „Wie oben, für compressore Nr.2“. A/M/B CO
  353 | Rotortemperatur Verdichter 3 „Wie oben, für den Verdichter Nr.3“. A/M/B CO | Rotortemperatur Verdichter 3 „Wie oben, für den Verdichter Nr.3“. A/M/B CO | Rotor temperature compressor 3 „Wie oben, für compressor Nr.3“. A/M/B CO | Rotor temperature compresseur 3 „Wie oben, für compresseur Nr.3“. A/M/B CO | Rotor temperature compressore 3 „Wie oben, für compressore Nr.3“. A/M/B CO
  354 | Rotortemperatur Verdichter 4 „Wie oben, für den Verdichter Nr.4“. A/M/B CO | Rotortemperatur Verdichter 4 „Wie oben, für den Verdichter Nr.4“. A/M/B CO | Rotor temperature compressor 4 „Wie oben, für compressor Nr.4“. A/M/B CO | Rotor temperature compresseur 4 „Wie oben, für compresseur Nr.4“. A/M/B CO | Rotor temperature compressore 4 „Wie oben, für compressore Nr.4“. A/M/B CO
  355 | Rotortemperatur Verdichter 5 „Wie oben, für den Verdichter Nr. 5“. A/M/B CO | Rotortemperatur Verdichter 5 „Wie oben, für den Verdichter Nr. 5“. A/M/B CO | Rotor temperature compressor 5 „Wie oben, für compressor Nr. 5“. A/M/B CO | Rotor temperature compresseur 5 „Wie oben, für compresseur Nr. 5“. A/M/B CO | Rotor temperature compressore 5 „Wie oben, für compressore Nr. 5“. A/M/B CO
  356 | Rotortemperatur Verdichter 6 „Wie oben, für den Verdichter Nr. 6“. A/M/B CO | Rotortemperatur Verdichter 6 „Wie oben, für den Verdichter Nr. 6“. A/M/B CO | Rotor temperature compressor 6 „Wie oben, für compressor Nr. 6“. A/M/B CO | Rotor temperature compresseur 6 „Wie oben, für compresseur Nr. 6“. A/M/B CO | Rotor temperature compressore 6 „Wie oben, für compressore Nr. 6“. A/M/B CO
  357 | Rotortemperatur Verdichter 7 „Wie oben, für den Verdichter Nr. 7“. A/M/B CO | Rotortemperatur Verdichter 7 „Wie oben, für den Verdichter Nr. 7“. A/M/B CO | Rotor temperature compressor 7 „Wie oben, für compressor Nr. 7“. A/M/B CO | Rotor temperature compresseur 7 „Wie oben, für compresseur Nr. 7“. A/M/B CO | Rotor temperature compressore 7 „Wie oben, für compressore Nr. 7“. A/M/B CO
  358 | Rotortemperatur Verdichter 8 „Wie oben, für den Verdichter Nr. 8“. A/M/B CO | Rotortemperatur Verdichter 8 „Wie oben, für den Verdichter Nr. 8“. A/M/B CO | Rotor temperature compressor 8 „Wie oben, für compressor Nr. 8“. A/M/B CO | Rotor temperature compresseur 8 „Wie oben, für compresseur Nr. 8“. A/M/B CO | Rotor temperature compressore 8 „Wie oben, für compressore Nr. 8“. A/M/B CO
  361 | Verdichtungsverhältnis Verdichter 1 Das Verdichtungsverhältnis des Verdichters Nr.1 ist höher als der zulässige Höchstwert (nur bei Einheiten mit Turbocor -Verdichtern). A/M/B CO | Verdichtungsverhältnis Verdichter 1 Das Verdichtungsverhältnis des Verdichters Nr.1 ist höher als der zulässige Höchstwert (nur bei Einheiten mit Turbocor -Verdichtern). A/M/B CO | Compression ratio compressor 1 Verdichtungsverhältnis compressors Nr.1 ist höher als zulässige Höchstwert (nur bei uniten mit Turbocor -compressorn). A/M/B CO | Compression ratio compresseur 1 Verdichtungsverhältnis compresseurs Nr.1 ist höher als zulässige Höchstwert (nur bei unitéen mit Turbocor -compresseurn). A/M/B CO | Compression ratio compressore 1 Verdichtungsverhältnis compressores Nr.1 ist höher als zulässige Höchstwert (nur bei unitàen mit Turbocor -compressoren). A/M/B CO
  362 | Verdichtungsverhältnis Verdichter 2 „Wie oben, für den Verdichter Nr.2“. A/M/B CO | Verdichtungsverhältnis Verdichter 2 „Wie oben, für den Verdichter Nr.2“. A/M/B CO | Compression ratio compressor 2 „Wie oben, für compressor Nr.2“. A/M/B CO | Compression ratio compresseur 2 „Wie oben, für compresseur Nr.2“. A/M/B CO | Compression ratio compressore 2 „Wie oben, für compressore Nr.2“. A/M/B CO
  363 | Verdichtungsverhältnis Verdichter 3 „Wie oben, für den Verdichter Nr.3“. A/M/B CO | Verdichtungsverhältnis Verdichter 3 „Wie oben, für den Verdichter Nr.3“. A/M/B CO | Compression ratio compressor 3 „Wie oben, für compressor Nr.3“. A/M/B CO | Compression ratio compresseur 3 „Wie oben, für compresseur Nr.3“. A/M/B CO | Compression ratio compressore 3 „Wie oben, für compressore Nr.3“. A/M/B CO
  364 | Verdichtungsverhältnis Verdichter 4 „Wie oben, für den Verdichter Nr.4“. A/M/B CO | Verdichtungsverhältnis Verdichter 4 „Wie oben, für den Verdichter Nr.4“. A/M/B CO | Compression ratio compressor 4 „Wie oben, für compressor Nr.4“. A/M/B CO | Compression ratio compresseur 4 „Wie oben, für compresseur Nr.4“. A/M/B CO | Compression ratio compressore 4 „Wie oben, für compressore Nr.4“. A/M/B CO
  365 | Verdichtungsverhältnis Verdichter 5 „Wie oben, für den Verdichter Nr. 5“. A/M/B CO | Verdichtungsverhältnis Verdichter 5 „Wie oben, für den Verdichter Nr. 5“. A/M/B CO | Compression ratio compressor 5 „Wie oben, für compressor Nr. 5“. A/M/B CO | Compression ratio compresseur 5 „Wie oben, für compresseur Nr. 5“. A/M/B CO | Compression ratio compressore 5 „Wie oben, für compressore Nr. 5“. A/M/B CO
  366 | Verdichtungsverhältnis Verdichter 6 „Wie oben, für den Verdichter Nr. 6“. A/M/B CO | Verdichtungsverhältnis Verdichter 6 „Wie oben, für den Verdichter Nr. 6“. A/M/B CO | Compression ratio compressor 6 „Wie oben, für compressor Nr. 6“. A/M/B CO | Compression ratio compresseur 6 „Wie oben, für compresseur Nr. 6“. A/M/B CO | Compression ratio compressore 6 „Wie oben, für compressore Nr. 6“. A/M/B CO
  367 | Verdichtungsverhältnis Verdichter 7 „Wie oben, für den Verdichter Nr. 7“. A/M/B CO | Verdichtungsverhältnis Verdichter 7 „Wie oben, für den Verdichter Nr. 7“. A/M/B CO | Compression ratio compressor 7 „Wie oben, für compressor Nr. 7“. A/M/B CO | Compression ratio compresseur 7 „Wie oben, für compresseur Nr. 7“. A/M/B CO | Compression ratio compressore 7 „Wie oben, für compressore Nr. 7“. A/M/B CO
  368 | Verdichtungsverhältnis Verdichter 8 „Wie oben, für den Verdichter Nr. 8“. A/M/B CO | Verdichtungsverhältnis Verdichter 8 „Wie oben, für den Verdichter Nr. 8“. A/M/B CO | Compression ratio compressor 8 „Wie oben, für compressor Nr. 8“. A/M/B CO | Compression ratio compresseur 8 „Wie oben, für compresseur Nr. 8“. A/M/B CO | Compression ratio compressore 8 „Wie oben, für compressore Nr. 8“. A/M/B CO
  371 | Lager Verdichter 1 Störung an den Lagern des Verdichters Nr.1 (nur bei Einheiten mit Turbocor -Verdichtern). A/M/B CO | Lager Verdichter 1 Störung an den Lagern des Verdichters Nr.1 (nur bei Einheiten mit Turbocor -Verdichtern). A/M/B CO | Compressor bearing 1 Störung an Lagern compressors Nr.1 (nur bei uniten mit Turbocor -compressorn). A/M/B CO | Compressor bearing 1 Störung an Lagern compresseurs Nr.1 (nur bei unitéen mit Turbocor -compresseurn). A/M/B CO | Compressor bearing 1 Störung an Lagern compressores Nr.1 (nur bei unitàen mit Turbocor -compressoren). A/M/B CO
  372 | Lager Verdichter 2 „Wie oben, für den Verdichter Nr.2“. A/M/B CO | Lager Verdichter 2 „Wie oben, für den Verdichter Nr.2“. A/M/B CO | Compressor bearing 2 „Wie oben, für compressor Nr.2“. A/M/B CO | Compressor bearing 2 „Wie oben, für compresseur Nr.2“. A/M/B CO | Compressor bearing 2 „Wie oben, für compressore Nr.2“. A/M/B CO
  373 | Lager Verdichter 3 „Wie oben, für den Verdichter Nr.3“. A/M/B CO | Lager Verdichter 3 „Wie oben, für den Verdichter Nr.3“. A/M/B CO | Compressor bearing 3 „Wie oben, für compressor Nr.3“. A/M/B CO | Compressor bearing 3 „Wie oben, für compresseur Nr.3“. A/M/B CO | Compressor bearing 3 „Wie oben, für compressore Nr.3“. A/M/B CO
  374 | Lager Verdichter 4 „Wie oben, für den Verdichter Nr.4“. A/M/B CO | Lager Verdichter 4 „Wie oben, für den Verdichter Nr.4“. A/M/B CO | Compressor bearing 4 „Wie oben, für compressor Nr.4“. A/M/B CO | Compressor bearing 4 „Wie oben, für compresseur Nr.4“. A/M/B CO | Compressor bearing 4 „Wie oben, für compressore Nr.4“. A/M/B CO
  375 | Lager Verdichter 5 „Wie oben, für den Verdichter Nr. 5“. A/M/B CO | Lager Verdichter 5 „Wie oben, für den Verdichter Nr. 5“. A/M/B CO | Compressor bearing 5 „Wie oben, für compressor Nr. 5“. A/M/B CO | Compressor bearing 5 „Wie oben, für compresseur Nr. 5“. A/M/B CO | Compressor bearing 5 „Wie oben, für compressore Nr. 5“. A/M/B CO
  376 | Lager Verdichter 6 „Wie oben, für den Verdichter Nr. 6“. A/M/B CO | Lager Verdichter 6 „Wie oben, für den Verdichter Nr. 6“. A/M/B CO | Compressor bearing 6 „Wie oben, für compressor Nr. 6“. A/M/B CO | Compressor bearing 6 „Wie oben, für compresseur Nr. 6“. A/M/B CO | Compressor bearing 6 „Wie oben, für compressore Nr. 6“. A/M/B CO
  377 | Lager Verdichter 7 „Wie oben, für den Verdichter Nr. 7“. A/M/B CO | Lager Verdichter 7 „Wie oben, für den Verdichter Nr. 7“. A/M/B CO | Compressor bearing 7 „Wie oben, für compressor Nr. 7“. A/M/B CO | Compressor bearing 7 „Wie oben, für compresseur Nr. 7“. A/M/B CO | Compressor bearing 7 „Wie oben, für compressore Nr. 7“. A/M/B CO
  378 | Lager Verdichter 8 „Wie oben, für den Verdichter Nr. 8“. A/M/B CO | Lager Verdichter 8 „Wie oben, für den Verdichter Nr. 8“. A/M/B CO | Compressor bearing 8 „Wie oben, für compressor Nr. 8“. A/M/B CO | Compressor bearing 8 „Wie oben, für compresseur Nr. 8“. A/M/B CO | Compressor bearing 8 „Wie oben, für compressore Nr. 8“. A/M/B CO
  381 | Temperatur SCR Verdichter 1 | Temperatur SCR Verdichter 1 | SCR temperature compressor 1 | SCR temperature compresseur 1 | SCR temperature compressore 1
  382 | Temperatur SCR Verdichter 2 „Wie oben, für den Verdichter Nr.2“. A/M/B CO | Temperatur SCR Verdichter 2 „Wie oben, für den Verdichter Nr.2“. A/M/B CO | SCR temperature compressor 2 „Wie oben, für compressor Nr.2“. A/M/B CO | SCR temperature compresseur 2 „Wie oben, für compresseur Nr.2“. A/M/B CO | SCR temperature compressore 2 „Wie oben, für compressore Nr.2“. A/M/B CO
  383 | Temperatur SCR Verdichter 3 „Wie oben, für den Verdichter Nr.3“. A/M/B CO | Temperatur SCR Verdichter 3 „Wie oben, für den Verdichter Nr.3“. A/M/B CO | SCR temperature compressor 3 „Wie oben, für compressor Nr.3“. A/M/B CO | SCR temperature compresseur 3 „Wie oben, für compresseur Nr.3“. A/M/B CO | SCR temperature compressore 3 „Wie oben, für compressore Nr.3“. A/M/B CO
  384 | Temperatur SCR Verdichter 4 „Wie oben, für den Verdichter Nr.4“. A/M/B CO | Temperatur SCR Verdichter 4 „Wie oben, für den Verdichter Nr.4“. A/M/B CO | SCR temperature compressor 4 „Wie oben, für compressor Nr.4“. A/M/B CO | SCR temperature compresseur 4 „Wie oben, für compresseur Nr.4“. A/M/B CO | SCR temperature compressore 4 „Wie oben, für compressore Nr.4“. A/M/B CO
  385 | Temperatur SCR Verdichter 5 „Wie oben, für den Verdichter Nr. 5“. A/M/B CO | Temperatur SCR Verdichter 5 „Wie oben, für den Verdichter Nr. 5“. A/M/B CO | SCR temperature compressor 5 „Wie oben, für compressor Nr. 5“. A/M/B CO | SCR temperature compresseur 5 „Wie oben, für compresseur Nr. 5“. A/M/B CO | SCR temperature compressore 5 „Wie oben, für compressore Nr. 5“. A/M/B CO
  386 | Temperatur SCR Verdichter 6 „Wie oben, für den Verdichter Nr. 6“. A/M/B CO | Temperatur SCR Verdichter 6 „Wie oben, für den Verdichter Nr. 6“. A/M/B CO | SCR temperature compressor 6 „Wie oben, für compressor Nr. 6“. A/M/B CO | SCR temperature compresseur 6 „Wie oben, für compresseur Nr. 6“. A/M/B CO | SCR temperature compressore 6 „Wie oben, für compressore Nr. 6“. A/M/B CO
  387 | Temperatur SCR Verdichter 7 „Wie oben, für den Verdichter Nr. 7“. A/M/B CO | Temperatur SCR Verdichter 7 „Wie oben, für den Verdichter Nr. 7“. A/M/B CO | SCR temperature compressor 7 „Wie oben, für compressor Nr. 7“. A/M/B CO | SCR temperature compresseur 7 „Wie oben, für compresseur Nr. 7“. A/M/B CO | SCR temperature compressore 7 „Wie oben, für compressore Nr. 7“. A/M/B CO
  388 | Temperatur SCR Verdichter 8 „Wie oben, für den Verdichter Nr. 8“. A/M/B CO | Temperatur SCR Verdichter 8 „Wie oben, für den Verdichter Nr. 8“. A/M/B CO | SCR temperature compressor 8 „Wie oben, für compressor Nr. 8“. A/M/B CO | SCR temperature compresseur 8 „Wie oben, für compresseur Nr. 8“. A/M/B CO | SCR temperature compressore 8 „Wie oben, für compressore Nr. 8“. A/M/B CO
  391 | Blockierung Rotor Verdichter 1 | Blockierung Rotor Verdichter 1 | Blockierung Rotor compressor 1 | Blockierung Rotor compresseur 1 | Blockierung Rotor compressore 1
  392 | Blockierung Rotor Verdichter 2 „Wie oben, für den Verdichter Nr.2“. A/M/B CO | Blockierung Rotor Verdichter 2 „Wie oben, für den Verdichter Nr.2“. A/M/B CO | Blockierung Rotor compressor 2 „Wie oben, für compressor Nr.2“. A/M/B CO | Blockierung Rotor compresseur 2 „Wie oben, für compresseur Nr.2“. A/M/B CO | Blockierung Rotor compressore 2 „Wie oben, für compressore Nr.2“. A/M/B CO
  393 | Blockierung Rotor Verdichter 3 „Wie oben, für den Verdichter Nr.3“. A/M/B CO | Blockierung Rotor Verdichter 3 „Wie oben, für den Verdichter Nr.3“. A/M/B CO | Blockierung Rotor compressor 3 „Wie oben, für compressor Nr.3“. A/M/B CO | Blockierung Rotor compresseur 3 „Wie oben, für compresseur Nr.3“. A/M/B CO | Blockierung Rotor compressore 3 „Wie oben, für compressore Nr.3“. A/M/B CO
  394 | Blockierung Rotor Verdichter 4 „Wie oben, für den Verdichter Nr.4“. A/M/B CO | Blockierung Rotor Verdichter 4 „Wie oben, für den Verdichter Nr.4“. A/M/B CO | Blockierung Rotor compressor 4 „Wie oben, für compressor Nr.4“. A/M/B CO | Blockierung Rotor compresseur 4 „Wie oben, für compresseur Nr.4“. A/M/B CO | Blockierung Rotor compressore 4 „Wie oben, für compressore Nr.4“. A/M/B CO
